KUKA KRL program: Inconel_dataset.src, Inconel_dataset.dat

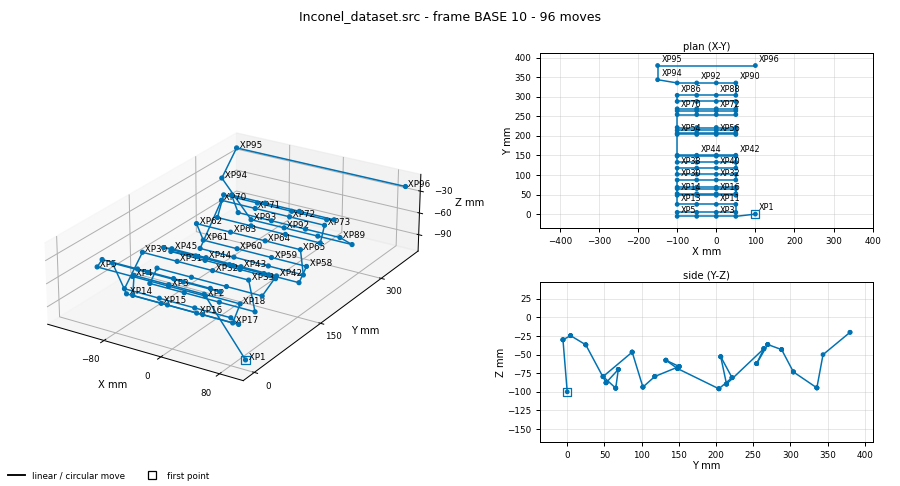
[picture p0: tool path of Inconel_dataset.src in frame BASE 10, 96 of 339 moves have a stored position in this frame; points joined in program order, loops and branches not executed]
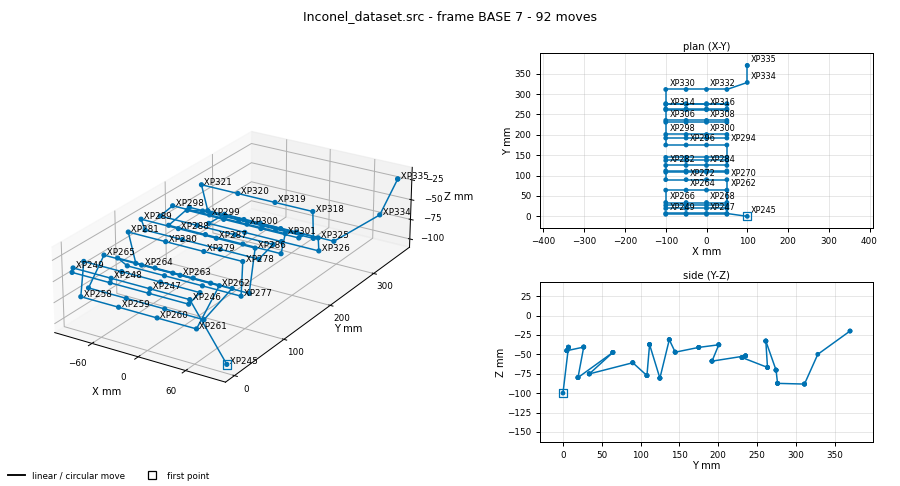
[picture p1: tool path of Inconel_dataset.src in frame BASE 7, 92 of 339 moves have a stored position in this frame; points joined in program order, loops and branches not executed]
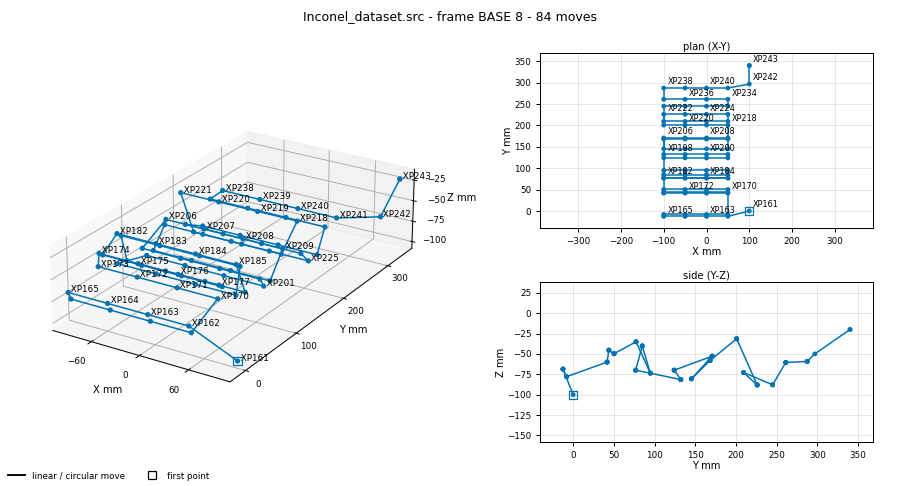
[picture p2: tool path of Inconel_dataset.src in frame BASE 8, 84 of 339 moves have a stored position in this frame; points joined in program order, loops and branches not executed]
--- Inconel_dataset.src ---
&ACCESS RVP1
&REL 1217
&PARAM WOPTRAJECTORYID = 2
&PARAM WOPTEMPLATENAME = WopCoreTemplatePath
&PARAM DISKPATH = KRC:\R1\Program\Working Paths
DEF  Inconel_dataset ( )

;FOLD INI
InitWopCoreSrc(#Init_Trajectory)
;ENDFOLD (INI)

;FOLD Manual mode
IF X_Rob_InManu THEN
;Write here the code executed only in manual mode

ENDIF
;ENDFOLD

X_Prod_En_Cours[2]=TRUE

;FOLD PTP PT_LoopPos1 Vel=10 % DEFAULT Tool[1]:Gun Base[0];%{PE}
;FOLD Parameters ;%{h}
;Params IlfProvider=kukaroboter.basistech.inlineforms.movement.old; Kuka.IsGlobalPoint=False; Kuka.PointName=PT_LoopPos1; Kuka.BlendingEnabled=False; Kuka.MoveDataPtpName=DEFAULT; Kuka.VelocityPtp=10; Kuka.CurrentCDSetIndex=0; Kuka.MovementParameterFieldEnabled=True; IlfCommand=PTP
;ENDFOLD
$BWDSTART = FALSE
PDAT_ACT = PDEFAULT
FDAT_ACT = FPT_LoopPos1
BAS(#PTP_PARAMS, 10.0)
SET_CD_PARAMS (0)
PTP XPT_LoopPos1
;ENDFOLD



;FOLD CHECK DAT-FILE GENERATION NUMBER
  IF APP_GENNUMBER <> 215375 THEN
    LOOP
      MsgQuit("InconsistenceSRCandDAT",,,,1)
      HALT
    ENDLOOP
  ENDIF
;ENDFOLD

;fold Jobinfo
;Job information: Inconel_dataset
;Product : 3.1.0.28784
;Date: 2026-09-10-16_16
;Project name: Inconel_dataset
;Author: Alhadi Zidan
;Company: CRITT-TJFU
;Division: CSAMProj
;Comment: Autogenerated CSAM Path
;endfold

; --- GLOBAL BLENDING OVERRIDES ---
$APO.CDIS = 1.0  ; Distance blending radius (mm)
$APO.CVEL = 100  ; Velocity blending (%)
$APO.CORI = 5.0  ; Orientation blending (degrees)
$ADVANCE = 5
;FOLD PTP P0 Vel=100 % P0 Tool[2] Base[10] ;%{PE}
;FOLD Parameters ;%{h}
;Params IlfProvider=kukaroboter.basistech.inlineforms.movement.old; Kuka.IsGlobalPoint=False; Kuka.PointName=P0; Kuka.BlendingEnabled=FALSE; Kuka.MoveDataName=PDATP0; Kuka.VelocityPath=100; Kuka.CurrentCDSetIndex=0; Kuka.MovementParameterFieldEnabled=True; IlfCommand=PTP
;ENDFOLD
$BWDSTART = FALSE
PDAT_ACT=PPDATP0
FDAT_ACT=FP0
BAS (#PTP_PARAMS,100)
SET_CD_PARAMS (0)
PTP XP0

;ENDFOLD
Routine_0()
Routine_1()
Routine_2()
Routine_3()
;FOLD PTP PT_LoopPos1 Vel=60 % DEFAULT Tool[1]:Gun Base[0];%{{PE}}
;FOLD Parameters ;%{{h}}
;Params IlfProvider=kukaroboter.basistech.inlineforms.movement.old; Kuka.IsGlobalPoint=False; Kuka.PointName=PT_LoopPos1; Kuka.BlendingEnabled=False; Kuka.MoveDataPtpName=DEFAULT; Kuka.VelocityPtp=10; Kuka.CurrentCDSetIndex=0; Kuka.MovementParameterFieldEnabled=True; IlfCommand=PTP
;ENDFOLD
$BWDSTART = FALSE
PDAT_ACT = PDEFAULT
FDAT_ACT = FPT_LoopPos1
BAS(#PTP_PARAMS, 60.0)
SET_CD_PARAMS (0)
PTP XPT_LoopPos1
;ENDFOLD
END

; --- Routine for substrate 0 ---
DEF Routine_0()
;FOLD LIN P1 CONT Vel=1.0 m/s CPDATP1 Tool[2] Base[10] ;%{PE}
;FOLD Parameters ;%{h}
;Params IlfProvider=kukaroboter.basistech.inlineforms.movement.old; Kuka.IsGlobalPoint=False; Kuka.PointName=P1; Kuka.BlendingEnabled=TRUE; Kuka.MoveDataName=CPDATP1; Kuka.VelocityPath=1.0; Kuka.CurrentCDSetIndex=0; Kuka.MovementParameterFieldEnabled=True; IlfCommand=LIN
;ENDFOLD
$BWDSTART = FALSE
LDAT_ACT=LCPDATP1
FDAT_ACT=FP1
BAS (#CP_PARAMS,1.0)
SET_CD_PARAMS (0)
LIN XP1 C_DIS

;ENDFOLD
;FOLD LIN P2 CONT Vel=0.116 m/s CPDATP2 Tool[2] Base[10] ;%{PE}
;FOLD Parameters ;%{h}
;Params IlfProvider=kukaroboter.basistech.inlineforms.movement.old; Kuka.IsGlobalPoint=False; Kuka.PointName=P2; Kuka.BlendingEnabled=TRUE; Kuka.MoveDataName=CPDATP2; Kuka.VelocityPath=0.116; Kuka.CurrentCDSetIndex=0; Kuka.MovementParameterFieldEnabled=True; IlfCommand=LIN
;ENDFOLD
$BWDSTART = FALSE
LDAT_ACT=LCPDATP2
FDAT_ACT=FP2
BAS (#CP_PARAMS,0.116)
SET_CD_PARAMS (0)
LIN XP2 C_DIS

;ENDFOLD
;FOLD LIN P3 CONT Vel=0.116 m/s CPDATP3 Tool[2] Base[10] ;%{PE}
;FOLD Parameters ;%{h}
;Params IlfProvider=kukaroboter.basistech.inlineforms.movement.old; Kuka.IsGlobalPoint=False; Kuka.PointName=P3; Kuka.BlendingEnabled=TRUE; Kuka.MoveDataName=CPDATP3; Kuka.VelocityPath=0.116; Kuka.CurrentCDSetIndex=0; Kuka.MovementParameterFieldEnabled=True; IlfCommand=LIN
;ENDFOLD
$BWDSTART = FALSE
LDAT_ACT=LCPDATP3
FDAT_ACT=FP3
BAS (#CP_PARAMS,0.116)
SET_CD_PARAMS (0)
LIN XP3 C_DIS

;ENDFOLD
;FOLD LIN P4 CONT Vel=0.116 m/s CPDATP4 Tool[2] Base[10] ;%{PE}
;FOLD Parameters ;%{h}
;Params IlfProvider=kukaroboter.basistech.inlineforms.movement.old; Kuka.IsGlobalPoint=False; Kuka.PointName=P4; Kuka.BlendingEnabled=TRUE; Kuka.MoveDataName=CPDATP4; Kuka.VelocityPath=0.116; Kuka.CurrentCDSetIndex=0; Kuka.MovementParameterFieldEnabled=True; IlfCommand=LIN
;ENDFOLD
$BWDSTART = FALSE
LDAT_ACT=LCPDATP4
FDAT_ACT=FP4
BAS (#CP_PARAMS,0.116)
SET_CD_PARAMS (0)
LIN XP4 C_DIS

;ENDFOLD
;FOLD LIN P5 CONT Vel=0.116 m/s CPDATP5 Tool[2] Base[10] ;%{PE}
;FOLD Parameters ;%{h}
;Params IlfProvider=kukaroboter.basistech.inlineforms.movement.old; Kuka.IsGlobalPoint=False; Kuka.PointName=P5; Kuka.BlendingEnabled=TRUE; Kuka.MoveDataName=CPDATP5; Kuka.VelocityPath=0.116; Kuka.CurrentCDSetIndex=0; Kuka.MovementParameterFieldEnabled=True; IlfCommand=LIN
;ENDFOLD
$BWDSTART = FALSE
LDAT_ACT=LCPDATP5
FDAT_ACT=FP5
BAS (#CP_PARAMS,0.116)
SET_CD_PARAMS (0)
LIN XP5 C_DIS

;ENDFOLD
;FOLD LIN P6 CONT Vel=0.099 m/s CPDATP6 Tool[2] Base[10] ;%{PE}
;FOLD Parameters ;%{h}
;Params IlfProvider=kukaroboter.basistech.inlineforms.movement.old; Kuka.IsGlobalPoint=False; Kuka.PointName=P6; Kuka.BlendingEnabled=TRUE; Kuka.MoveDataName=CPDATP6; Kuka.VelocityPath=0.099; Kuka.CurrentCDSetIndex=0; Kuka.MovementParameterFieldEnabled=True; IlfCommand=LIN
;ENDFOLD
$BWDSTART = FALSE
LDAT_ACT=LCPDATP6
FDAT_ACT=FP6
BAS (#CP_PARAMS,0.099)
SET_CD_PARAMS (0)
LIN XP6 C_DIS

;ENDFOLD
;FOLD LIN P7 CONT Vel=0.099 m/s CPDATP7 Tool[2] Base[10] ;%{PE}
;FOLD Parameters ;%{h}
;Params IlfProvider=kukaroboter.basistech.inlineforms.movement.old; Kuka.IsGlobalPoint=False; Kuka.PointName=P7; Kuka.BlendingEnabled=TRUE; Kuka.MoveDataName=CPDATP7; Kuka.VelocityPath=0.099; Kuka.CurrentCDSetIndex=0; Kuka.MovementParameterFieldEnabled=True; IlfCommand=LIN
;ENDFOLD
$BWDSTART = FALSE
LDAT_ACT=LCPDATP7
FDAT_ACT=FP7
BAS (#CP_PARAMS,0.099)
SET_CD_PARAMS (0)
LIN XP7 C_DIS

;ENDFOLD
;FOLD LIN P8 CONT Vel=0.099 m/s CPDATP8 Tool[2] Base[10] ;%{PE}
;FOLD Parameters ;%{h}
;Params IlfProvider=kukaroboter.basistech.inlineforms.movement.old; Kuka.IsGlobalPoint=False; Kuka.PointName=P8; Kuka.BlendingEnabled=TRUE; Kuka.MoveDataName=CPDATP8; Kuka.VelocityPath=0.099; Kuka.CurrentCDSetIndex=0; Kuka.MovementParameterFieldEnabled=True; IlfCommand=LIN
;ENDFOLD
$BWDSTART = FALSE
LDAT_ACT=LCPDATP8
FDAT_ACT=FP8
BAS (#CP_PARAMS,0.099)
SET_CD_PARAMS (0)
LIN XP8 C_DIS

;ENDFOLD
;FOLD LIN P9 CONT Vel=0.099 m/s CPDATP9 Tool[2] Base[10] ;%{PE}
;FOLD Parameters ;%{h}
;Params IlfProvider=kukaroboter.basistech.inlineforms.movement.old; Kuka.IsGlobalPoint=False; Kuka.PointName=P9; Kuka.BlendingEnabled=TRUE; Kuka.MoveDataName=CPDATP9; Kuka.VelocityPath=0.099; Kuka.CurrentCDSetIndex=0; Kuka.MovementParameterFieldEnabled=True; IlfCommand=LIN
;ENDFOLD
$BWDSTART = FALSE
LDAT_ACT=LCPDATP9
FDAT_ACT=FP9
BAS (#CP_PARAMS,0.099)
SET_CD_PARAMS (0)
LIN XP9 C_DIS

;ENDFOLD
;FOLD LIN P10 CONT Vel=0.075 m/s CPDATP10 Tool[2] Base[10] ;%{PE}
;FOLD Parameters ;%{h}
;Params IlfProvider=kukaroboter.basistech.inlineforms.movement.old; Kuka.IsGlobalPoint=False; Kuka.PointName=P10; Kuka.BlendingEnabled=TRUE; Kuka.MoveDataName=CPDATP10; Kuka.VelocityPath=0.075; Kuka.CurrentCDSetIndex=0; Kuka.MovementParameterFieldEnabled=True; IlfCommand=LIN
;ENDFOLD
$BWDSTART = FALSE
LDAT_ACT=LCPDATP10
FDAT_ACT=FP10
BAS (#CP_PARAMS,0.075)
SET_CD_PARAMS (0)
LIN XP10 C_DIS

;ENDFOLD
;FOLD LIN P11 CONT Vel=0.075 m/s CPDATP11 Tool[2] Base[10] ;%{PE}
;FOLD Parameters ;%{h}
;Params IlfProvider=kukaroboter.basistech.inlineforms.movement.old; Kuka.IsGlobalPoint=False; Kuka.PointName=P11; Kuka.BlendingEnabled=TRUE; Kuka.MoveDataName=CPDATP11; Kuka.VelocityPath=0.075; Kuka.CurrentCDSetIndex=0; Kuka.MovementParameterFieldEnabled=True; IlfCommand=LIN
;ENDFOLD
$BWDSTART = FALSE
LDAT_ACT=LCPDATP11
FDAT_ACT=FP11
BAS (#CP_PARAMS,0.075)
SET_CD_PARAMS (0)
LIN XP11 C_DIS

;ENDFOLD
;FOLD LIN P12 CONT Vel=0.075 m/s CPDATP12 Tool[2] Base[10] ;%{PE}
;FOLD Parameters ;%{h}
;Params IlfProvider=kukaroboter.basistech.inlineforms.movement.old; Kuka.IsGlobalPoint=False; Kuka.PointName=P12; Kuka.BlendingEnabled=TRUE; Kuka.MoveDataName=CPDATP12; Kuka.VelocityPath=0.075; Kuka.CurrentCDSetIndex=0; Kuka.MovementParameterFieldEnabled=True; IlfCommand=LIN
;ENDFOLD
$BWDSTART = FALSE
LDAT_ACT=LCPDATP12
FDAT_ACT=FP12
BAS (#CP_PARAMS,0.075)
SET_CD_PARAMS (0)
LIN XP12 C_DIS

;ENDFOLD
;FOLD LIN P13 CONT Vel=0.075 m/s CPDATP13 Tool[2] Base[10] ;%{PE}
;FOLD Parameters ;%{h}
;Params IlfProvider=kukaroboter.basistech.inlineforms.movement.old; Kuka.IsGlobalPoint=False; Kuka.PointName=P13; Kuka.BlendingEnabled=TRUE; Kuka.MoveDataName=CPDATP13; Kuka.VelocityPath=0.075; Kuka.CurrentCDSetIndex=0; Kuka.MovementParameterFieldEnabled=True; IlfCommand=LIN
;ENDFOLD
$BWDSTART = FALSE
LDAT_ACT=LCPDATP13
FDAT_ACT=FP13
BAS (#CP_PARAMS,0.075)
SET_CD_PARAMS (0)
LIN XP13 C_DIS

;ENDFOLD
;FOLD LIN P14 CONT Vel=0.113 m/s CPDATP14 Tool[2] Base[10] ;%{PE}
;FOLD Parameters ;%{h}
;Params IlfProvider=kukaroboter.basistech.inlineforms.movement.old; Kuka.IsGlobalPoint=False; Kuka.PointName=P14; Kuka.BlendingEnabled=TRUE; Kuka.MoveDataName=CPDATP14; Kuka.VelocityPath=0.113; Kuka.CurrentCDSetIndex=0; Kuka.MovementParameterFieldEnabled=True; IlfCommand=LIN
;ENDFOLD
$BWDSTART = FALSE
LDAT_ACT=LCPDATP14
FDAT_ACT=FP14
BAS (#CP_PARAMS,0.113)
SET_CD_PARAMS (0)
LIN XP14 C_DIS

;ENDFOLD
;FOLD LIN P15 CONT Vel=0.113 m/s CPDATP15 Tool[2] Base[10] ;%{PE}
;FOLD Parameters ;%{h}
;Params IlfProvider=kukaroboter.basistech.inlineforms.movement.old; Kuka.IsGlobalPoint=False; Kuka.PointName=P15; Kuka.BlendingEnabled=TRUE; Kuka.MoveDataName=CPDATP15; Kuka.VelocityPath=0.113; Kuka.CurrentCDSetIndex=0; Kuka.MovementParameterFieldEnabled=True; IlfCommand=LIN
;ENDFOLD
$BWDSTART = FALSE
LDAT_ACT=LCPDATP15
FDAT_ACT=FP15
BAS (#CP_PARAMS,0.113)
SET_CD_PARAMS (0)
LIN XP15 C_DIS

;ENDFOLD
;FOLD LIN P16 CONT Vel=0.113 m/s CPDATP16 Tool[2] Base[10] ;%{PE}
;FOLD Parameters ;%{h}
;Params IlfProvider=kukaroboter.basistech.inlineforms.movement.old; Kuka.IsGlobalPoint=False; Kuka.PointName=P16; Kuka.BlendingEnabled=TRUE; Kuka.MoveDataName=CPDATP16; Kuka.VelocityPath=0.113; Kuka.CurrentCDSetIndex=0; Kuka.MovementParameterFieldEnabled=True; IlfCommand=LIN
;ENDFOLD
$BWDSTART = FALSE
LDAT_ACT=LCPDATP16
FDAT_ACT=FP16
BAS (#CP_PARAMS,0.113)
SET_CD_PARAMS (0)
LIN XP16 C_DIS

;ENDFOLD
;FOLD LIN P17 CONT Vel=0.113 m/s CPDATP17 Tool[2] Base[10] ;%{PE}
;FOLD Parameters ;%{h}
;Params IlfProvider=kukaroboter.basistech.inlineforms.movement.old; Kuka.IsGlobalPoint=False; Kuka.PointName=P17; Kuka.BlendingEnabled=TRUE; Kuka.MoveDataName=CPDATP17; Kuka.VelocityPath=0.113; Kuka.CurrentCDSetIndex=0; Kuka.MovementParameterFieldEnabled=True; IlfCommand=LIN
;ENDFOLD
$BWDSTART = FALSE
LDAT_ACT=LCPDATP17
FDAT_ACT=FP17
BAS (#CP_PARAMS,0.113)
SET_CD_PARAMS (0)
LIN XP17 C_DIS

;ENDFOLD
;FOLD LIN P18 CONT Vel=0.086 m/s CPDATP18 Tool[2] Base[10] ;%{PE}
;FOLD Parameters ;%{h}
;Params IlfProvider=kukaroboter.basistech.inlineforms.movement.old; Kuka.IsGlobalPoint=False; Kuka.PointName=P18; Kuka.BlendingEnabled=TRUE; Kuka.MoveDataName=CPDATP18; Kuka.VelocityPath=0.086; Kuka.CurrentCDSetIndex=0; Kuka.MovementParameterFieldEnabled=True; IlfCommand=LIN
;ENDFOLD
$BWDSTART = FALSE
LDAT_ACT=LCPDATP18
FDAT_ACT=FP18
BAS (#CP_PARAMS,0.086)
SET_CD_PARAMS (0)
LIN XP18 C_DIS

;ENDFOLD
;FOLD LIN P19 CONT Vel=0.086 m/s CPDATP19 Tool[2] Base[10] ;%{PE}
;FOLD Parameters ;%{h}
;Params IlfProvider=kukaroboter.basistech.inlineforms.movement.old; Kuka.IsGlobalPoint=False; Kuka.PointName=P19; Kuka.BlendingEnabled=TRUE; Kuka.MoveDataName=CPDATP19; Kuka.VelocityPath=0.086; Kuka.CurrentCDSetIndex=0; Kuka.MovementParameterFieldEnabled=True; IlfCommand=LIN
;ENDFOLD
$BWDSTART = FALSE
LDAT_ACT=LCPDATP19
FDAT_ACT=FP19
BAS (#CP_PARAMS,0.086)
SET_CD_PARAMS (0)
LIN XP19 C_DIS

;ENDFOLD
;FOLD LIN P20 CONT Vel=0.086 m/s CPDATP20 Tool[2] Base[10] ;%{PE}
;FOLD Parameters ;%{h}
;Params IlfProvider=kukaroboter.basistech.inlineforms.movement.old; Kuka.IsGlobalPoint=False; Kuka.PointName=P20; Kuka.BlendingEnabled=TRUE; Kuka.MoveDataName=CPDATP20; Kuka.VelocityPath=0.086; Kuka.CurrentCDSetIndex=0; Kuka.MovementParameterFieldEnabled=True; IlfCommand=LIN
;ENDFOLD
$BWDSTART = FALSE
LDAT_ACT=LCPDATP20
FDAT_ACT=FP20
BAS (#CP_PARAMS,0.086)
SET_CD_PARAMS (0)
LIN XP20 C_DIS

;ENDFOLD
;FOLD LIN P21 CONT Vel=0.086 m/s CPDATP21 Tool[2] Base[10] ;%{PE}
;FOLD Parameters ;%{h}
;Params IlfProvider=kukaroboter.basistech.inlineforms.movement.old; Kuka.IsGlobalPoint=False; Kuka.PointName=P21; Kuka.BlendingEnabled=TRUE; Kuka.MoveDataName=CPDATP21; Kuka.VelocityPath=0.086; Kuka.CurrentCDSetIndex=0; Kuka.MovementParameterFieldEnabled=True; IlfCommand=LIN
;ENDFOLD
$BWDSTART = FALSE
LDAT_ACT=LCPDATP21
FDAT_ACT=FP21
BAS (#CP_PARAMS,0.086)
SET_CD_PARAMS (0)
LIN XP21 C_DIS

;ENDFOLD
;FOLD LIN P22 CONT Vel=0.073 m/s CPDATP22 Tool[2] Base[10] ;%{PE}
;FOLD Parameters ;%{h}
;Params IlfProvider=kukaroboter.basistech.inlineforms.movement.old; Kuka.IsGlobalPoint=False; Kuka.PointName=P22; Kuka.BlendingEnabled=TRUE; Kuka.MoveDataName=CPDATP22; Kuka.VelocityPath=0.073; Kuka.CurrentCDSetIndex=0; Kuka.MovementParameterFieldEnabled=True; IlfCommand=LIN
;ENDFOLD
$BWDSTART = FALSE
LDAT_ACT=LCPDATP22
FDAT_ACT=FP22
BAS (#CP_PARAMS,0.073)
SET_CD_PARAMS (0)
LIN XP22 C_DIS

;ENDFOLD
;FOLD LIN P23 CONT Vel=0.073 m/s CPDATP23 Tool[2] Base[10] ;%{PE}
;FOLD Parameters ;%{h}
;Params IlfProvider=kukaroboter.basistech.inlineforms.movement.old; Kuka.IsGlobalPoint=False; Kuka.PointName=P23; Kuka.BlendingEnabled=TRUE; Kuka.MoveDataName=CPDATP23; Kuka.VelocityPath=0.073; Kuka.CurrentCDSetIndex=0; Kuka.MovementParameterFieldEnabled=True; IlfCommand=LIN
;ENDFOLD
$BWDSTART = FALSE
LDAT_ACT=LCPDATP23
FDAT_ACT=FP23
BAS (#CP_PARAMS,0.073)
SET_CD_PARAMS (0)
LIN XP23 C_DIS

;ENDFOLD
;FOLD LIN P24 CONT Vel=0.073 m/s CPDATP24 Tool[2] Base[10] ;%{PE}
;FOLD Parameters ;%{h}
;Params IlfProvider=kukaroboter.basistech.inlineforms.movement.old; Kuka.IsGlobalPoint=False; Kuka.PointName=P24; Kuka.BlendingEnabled=TRUE; Kuka.MoveDataName=CPDATP24; Kuka.VelocityPath=0.073; Kuka.CurrentCDSetIndex=0; Kuka.MovementParameterFieldEnabled=True; IlfCommand=LIN
;ENDFOLD
$BWDSTART = FALSE
LDAT_ACT=LCPDATP24
FDAT_ACT=FP24
BAS (#CP_PARAMS,0.073)
SET_CD_PARAMS (0)
LIN XP24 C_DIS

;ENDFOLD
;FOLD LIN P25 CONT Vel=0.073 m/s CPDATP25 Tool[2] Base[10] ;%{PE}
;FOLD Parameters ;%{h}
;Params IlfProvider=kukaroboter.basistech.inlineforms.movement.old; Kuka.IsGlobalPoint=False; Kuka.PointName=P25; Kuka.BlendingEnabled=TRUE; Kuka.MoveDataName=CPDATP25; Kuka.VelocityPath=0.073; Kuka.CurrentCDSetIndex=0; Kuka.MovementParameterFieldEnabled=True; IlfCommand=LIN
;ENDFOLD
$BWDSTART = FALSE
LDAT_ACT=LCPDATP25
FDAT_ACT=FP25
BAS (#CP_PARAMS,0.073)
SET_CD_PARAMS (0)
LIN XP25 C_DIS

;ENDFOLD
;FOLD LIN P26 CONT Vel=0.137 m/s CPDATP26 Tool[2] Base[10] ;%{PE}
;FOLD Parameters ;%{h}
;Params IlfProvider=kukaroboter.basistech.inlineforms.movement.old; Kuka.IsGlobalPoint=False; Kuka.PointName=P26; Kuka.BlendingEnabled=TRUE; Kuka.MoveDataName=CPDATP26; Kuka.VelocityPath=0.137; Kuka.CurrentCDSetIndex=0; Kuka.MovementParameterFieldEnabled=True; IlfCommand=LIN
;ENDFOLD
$BWDSTART = FALSE
LDAT_ACT=LCPDATP26
FDAT_ACT=FP26
BAS (#CP_PARAMS,0.137)
SET_CD_PARAMS (0)
LIN XP26 C_DIS

;ENDFOLD
;FOLD LIN P27 CONT Vel=0.137 m/s CPDATP27 Tool[2] Base[10] ;%{PE}
;FOLD Parameters ;%{h}
;Params IlfProvider=kukaroboter.basistech.inlineforms.movement.old; Kuka.IsGlobalPoint=False; Kuka.PointName=P27; Kuka.BlendingEnabled=TRUE; Kuka.MoveDataName=CPDATP27; Kuka.VelocityPath=0.137; Kuka.CurrentCDSetIndex=0; Kuka.MovementParameterFieldEnabled=True; IlfCommand=LIN
;ENDFOLD
$BWDSTART = FALSE
LDAT_ACT=LCPDATP27
FDAT_ACT=FP27
BAS (#CP_PARAMS,0.137)
SET_CD_PARAMS (0)
LIN XP27 C_DIS

;ENDFOLD
;FOLD LIN P28 CONT Vel=0.137 m/s CPDATP28 Tool[2] Base[10] ;%{PE}
;FOLD Parameters ;%{h}
;Params IlfProvider=kukaroboter.basistech.inlineforms.movement.old; Kuka.IsGlobalPoint=False; Kuka.PointName=P28; Kuka.BlendingEnabled=TRUE; Kuka.MoveDataName=CPDATP28; Kuka.VelocityPath=0.137; Kuka.CurrentCDSetIndex=0; Kuka.MovementParameterFieldEnabled=True; IlfCommand=LIN
;ENDFOLD
$BWDSTART = FALSE
LDAT_ACT=LCPDATP28
FDAT_ACT=FP28
BAS (#CP_PARAMS,0.137)
SET_CD_PARAMS (0)
LIN XP28 C_DIS

;ENDFOLD
;FOLD LIN P29 CONT Vel=0.137 m/s CPDATP29 Tool[2] Base[10] ;%{PE}
;FOLD Parameters ;%{h}
;Params IlfProvider=kukaroboter.basistech.inlineforms.movement.old; Kuka.IsGlobalPoint=False; Kuka.PointName=P29; Kuka.BlendingEnabled=TRUE; Kuka.MoveDataName=CPDATP29; Kuka.VelocityPath=0.137; Kuka.CurrentCDSetIndex=0; Kuka.MovementParameterFieldEnabled=True; IlfCommand=LIN
;ENDFOLD
$BWDSTART = FALSE
LDAT_ACT=LCPDATP29
FDAT_ACT=FP29
BAS (#CP_PARAMS,0.137)
SET_CD_PARAMS (0)
LIN XP29 C_DIS

;ENDFOLD
;FOLD LIN P30 CONT Vel=0.082 m/s CPDATP30 Tool[2] Base[10] ;%{PE}
;FOLD Parameters ;%{h}
;Params IlfProvider=kukaroboter.basistech.inlineforms.movement.old; Kuka.IsGlobalPoint=False; Kuka.PointName=P30; Kuka.BlendingEnabled=TRUE; Kuka.MoveDataName=CPDATP30; Kuka.VelocityPath=0.082; Kuka.CurrentCDSetIndex=0; Kuka.MovementParameterFieldEnabled=True; IlfCommand=LIN
;ENDFOLD
$BWDSTART = FALSE
LDAT_ACT=LCPDATP30
FDAT_ACT=FP30
BAS (#CP_PARAMS,0.082)
SET_CD_PARAMS (0)
LIN XP30 C_DIS

;ENDFOLD
;FOLD LIN P31 CONT Vel=0.082 m/s CPDATP31 Tool[2] Base[10] ;%{PE}
;FOLD Parameters ;%{h}
;Params IlfProvider=kukaroboter.basistech.inlineforms.movement.old; Kuka.IsGlobalPoint=False; Kuka.PointName=P31; Kuka.BlendingEnabled=TRUE; Kuka.MoveDataName=CPDATP31; Kuka.VelocityPath=0.082; Kuka.CurrentCDSetIndex=0; Kuka.MovementParameterFieldEnabled=True; IlfCommand=LIN
;ENDFOLD
$BWDSTART = FALSE
LDAT_ACT=LCPDATP31
FDAT_ACT=FP31
BAS (#CP_PARAMS,0.082)
SET_CD_PARAMS (0)
LIN XP31 C_DIS

;ENDFOLD
;FOLD LIN P32 CONT Vel=0.082 m/s CPDATP32 Tool[2] Base[10] ;%{PE}
;FOLD Parameters ;%{h}
;Params IlfProvider=kukaroboter.basistech.inlineforms.movement.old; Kuka.IsGlobalPoint=False; Kuka.PointName=P32; Kuka.BlendingEnabled=TRUE; Kuka.MoveDataName=CPDATP32; Kuka.VelocityPath=0.082; Kuka.CurrentCDSetIndex=0; Kuka.MovementParameterFieldEnabled=True; IlfCommand=LIN
;ENDFOLD
$BWDSTART = FALSE
LDAT_ACT=LCPDATP32
FDAT_ACT=FP32
BAS (#CP_PARAMS,0.082)
SET_CD_PARAMS (0)
LIN XP32 C_DIS

;ENDFOLD
;FOLD LIN P33 CONT Vel=0.082 m/s CPDATP33 Tool[2] Base[10] ;%{PE}
;FOLD Parameters ;%{h}
;Params IlfProvider=kukaroboter.basistech.inlineforms.movement.old; Kuka.IsGlobalPoint=False; Kuka.PointName=P33; Kuka.BlendingEnabled=TRUE; Kuka.MoveDataName=CPDATP33; Kuka.VelocityPath=0.082; Kuka.CurrentCDSetIndex=0; Kuka.MovementParameterFieldEnabled=True; IlfCommand=LIN
;ENDFOLD
$BWDSTART = FALSE
LDAT_ACT=LCPDATP33
FDAT_ACT=FP33
BAS (#CP_PARAMS,0.082)
SET_CD_PARAMS (0)
LIN XP33 C_DIS

;ENDFOLD
;FOLD LIN P34 CONT Vel=0.086 m/s CPDATP34 Tool[2] Base[10] ;%{PE}
;FOLD Parameters ;%{h}
;Params IlfProvider=kukaroboter.basistech.inlineforms.movement.old; Kuka.IsGlobalPoint=False; Kuka.PointName=P34; Kuka.BlendingEnabled=TRUE; Kuka.MoveDataName=CPDATP34; Kuka.VelocityPath=0.086; Kuka.CurrentCDSetIndex=0; Kuka.MovementParameterFieldEnabled=True; IlfCommand=LIN
;ENDFOLD
$BWDSTART = FALSE
LDAT_ACT=LCPDATP34
FDAT_ACT=FP34
BAS (#CP_PARAMS,0.086)
SET_CD_PARAMS (0)
LIN XP34 C_DIS

;ENDFOLD
;FOLD LIN P35 CONT Vel=0.086 m/s CPDATP35 Tool[2] Base[10] ;%{PE}
;FOLD Parameters ;%{h}
;Params IlfProvider=kukaroboter.basistech.inlineforms.movement.old; Kuka.IsGlobalPoint=False; Kuka.PointName=P35; Kuka.BlendingEnabled=TRUE; Kuka.MoveDataName=CPDATP35; Kuka.VelocityPath=0.086; Kuka.CurrentCDSetIndex=0; Kuka.MovementParameterFieldEnabled=True; IlfCommand=LIN
;ENDFOLD
$BWDSTART = FALSE
LDAT_ACT=LCPDATP35
FDAT_ACT=FP35
BAS (#CP_PARAMS,0.086)
SET_CD_PARAMS (0)
LIN XP35 C_DIS

;ENDFOLD
;FOLD LIN P36 CONT Vel=0.086 m/s CPDATP36 Tool[2] Base[10] ;%{PE}
;FOLD Parameters ;%{h}
;Params IlfProvider=kukaroboter.basistech.inlineforms.movement.old; Kuka.IsGlobalPoint=False; Kuka.PointName=P36; Kuka.BlendingEnabled=TRUE; Kuka.MoveDataName=CPDATP36; Kuka.VelocityPath=0.086; Kuka.CurrentCDSetIndex=0; Kuka.MovementParameterFieldEnabled=True; IlfCommand=LIN
;ENDFOLD
$BWDSTART = FALSE
LDAT_ACT=LCPDATP36
FDAT_ACT=FP36
BAS (#CP_PARAMS,0.086)
SET_CD_PARAMS (0)
LIN XP36 C_DIS

;ENDFOLD
;FOLD LIN P37 CONT Vel=0.086 m/s CPDATP37 Tool[2] Base[10] ;%{PE}
;FOLD Parameters ;%{h}
;Params IlfProvider=kukaroboter.basistech.inlineforms.movement.old; Kuka.IsGlobalPoint=False; Kuka.PointName=P37; Kuka.BlendingEnabled=TRUE; Kuka.MoveDataName=CPDATP37; Kuka.VelocityPath=0.086; Kuka.CurrentCDSetIndex=0; Kuka.MovementParameterFieldEnabled=True; IlfCommand=LIN
;ENDFOLD
$BWDSTART = FALSE
LDAT_ACT=LCPDATP37
FDAT_ACT=FP37
BAS (#CP_PARAMS,0.086)
SET_CD_PARAMS (0)
LIN XP37 C_DIS

;ENDFOLD
;FOLD LIN P38 CONT Vel=0.097 m/s CPDATP38 Tool[2] Base[10] ;%{PE}
;FOLD Parameters ;%{h}
;Params IlfProvider=kukaroboter.basistech.inlineforms.movement.old; Kuka.IsGlobalPoint=False; Kuka.PointName=P38; Kuka.BlendingEnabled=TRUE; Kuka.MoveDataName=CPDATP38; Kuka.VelocityPath=0.097; Kuka.CurrentCDSetIndex=0; Kuka.MovementParameterFieldEnabled=True; IlfCommand=LIN
;ENDFOLD
$BWDSTART = FALSE
LDAT_ACT=LCPDATP38
FDAT_ACT=FP38
BAS (#CP_PARAMS,0.097)
SET_CD_PARAMS (0)
LIN XP38 C_DIS

;ENDFOLD
;FOLD LIN P39 CONT Vel=0.097 m/s CPDATP39 Tool[2] Base[10] ;%{PE}
;FOLD Parameters ;%{h}
;Params IlfProvider=kukaroboter.basistech.inlineforms.movement.old; Kuka.IsGlobalPoint=False; Kuka.PointName=P39; Kuka.BlendingEnabled=TRUE; Kuka.MoveDataName=CPDATP39; Kuka.VelocityPath=0.097; Kuka.CurrentCDSetIndex=0; Kuka.MovementParameterFieldEnabled=True; IlfCommand=LIN
;ENDFOLD
$BWDSTART = FALSE
LDAT_ACT=LCPDATP39
FDAT_ACT=FP39
BAS (#CP_PARAMS,0.097)
SET_CD_PARAMS (0)
LIN XP39 C_DIS

;ENDFOLD
;FOLD LIN P40 CONT Vel=0.097 m/s CPDATP40 Tool[2] Base[10] ;%{PE}
;FOLD Parameters ;%{h}
;Params IlfProvider=kukaroboter.basistech.inlineforms.movement.old; Kuka.IsGlobalPoint=False; Kuka.PointName=P40; Kuka.BlendingEnabled=TRUE; Kuka.MoveDataName=CPDATP40; Kuka.VelocityPath=0.097; Kuka.CurrentCDSetIndex=0; Kuka.MovementParameterFieldEnabled=True; IlfCommand=LIN
;ENDFOLD
$BWDSTART = FALSE
LDAT_ACT=LCPDATP40
FDAT_ACT=FP40
BAS (#CP_PARAMS,0.097)
SET_CD_PARAMS (0)
LIN XP40 C_DIS

;ENDFOLD
;FOLD LIN P41 CONT Vel=0.097 m/s CPDATP41 Tool[2] Base[10] ;%{PE}
;FOLD Parameters ;%{h}
;Params IlfProvider=kukaroboter.basistech.inlineforms.movement.old; Kuka.IsGlobalPoint=False; Kuka.PointName=P41; Kuka.BlendingEnabled=TRUE; Kuka.MoveDataName=CPDATP41; Kuka.VelocityPath=0.097; Kuka.CurrentCDSetIndex=0; Kuka.MovementParameterFieldEnabled=True; IlfCommand=LIN
;ENDFOLD
$BWDSTART = FALSE
LDAT_ACT=LCPDATP41
FDAT_ACT=FP41
BAS (#CP_PARAMS,0.097)
SET_CD_PARAMS (0)
LIN XP41 C_DIS

;ENDFOLD
;FOLD LIN P42 CONT Vel=0.136 m/s CPDATP42 Tool[2] Base[10] ;%{PE}
;FOLD Parameters ;%{h}
;Params IlfProvider=kukaroboter.basistech.inlineforms.movement.old; Kuka.IsGlobalPoint=False; Kuka.PointName=P42; Kuka.BlendingEnabled=TRUE; Kuka.MoveDataName=CPDATP42; Kuka.VelocityPath=0.136; Kuka.CurrentCDSetIndex=0; Kuka.MovementParameterFieldEnabled=True; IlfCommand=LIN
;ENDFOLD
$BWDSTART = FALSE
LDAT_ACT=LCPDATP42
FDAT_ACT=FP42
BAS (#CP_PARAMS,0.136)
SET_CD_PARAMS (0)
LIN XP42 C_DIS

;ENDFOLD
;FOLD LIN P43 CONT Vel=0.136 m/s CPDATP43 Tool[2] Base[10] ;%{PE}
;FOLD Parameters ;%{h}
;Params IlfProvider=kukaroboter.basistech.inlineforms.movement.old; Kuka.IsGlobalPoint=False; Kuka.PointName=P43; Kuka.BlendingEnabled=TRUE; Kuka.MoveDataName=CPDATP43; Kuka.VelocityPath=0.136; Kuka.CurrentCDSetIndex=0; Kuka.MovementParameterFieldEnabled=True; IlfCommand=LIN
;ENDFOLD
$BWDSTART = FALSE
LDAT_ACT=LCPDATP43
FDAT_ACT=FP43
BAS (#CP_PARAMS,0.136)
SET_CD_PARAMS (0)
LIN XP43 C_DIS

;ENDFOLD
;FOLD LIN P44 CONT Vel=0.136 m/s CPDATP44 Tool[2] Base[10] ;%{PE}
;FOLD Parameters ;%{h}
;Params IlfProvider=kukaroboter.basistech.inlineforms.movement.old; Kuka.IsGlobalPoint=False; Kuka.PointName=P44; Kuka.BlendingEnabled=TRUE; Kuka.MoveDataName=CPDATP44; Kuka.VelocityPath=0.136; Kuka.CurrentCDSetIndex=0; Kuka.MovementParameterFieldEnabled=True; IlfCommand=LIN
;ENDFOLD
$BWDSTART = FALSE
LDAT_ACT=LCPDATP44
FDAT_ACT=FP44
BAS (#CP_PARAMS,0.136)
SET_CD_PARAMS (0)
LIN XP44 C_DIS

;ENDFOLD
;FOLD LIN P45 CONT Vel=0.136 m/s CPDATP45 Tool[2] Base[10] ;%{PE}
;FOLD Parameters ;%{h}
;Params IlfProvider=kukaroboter.basistech.inlineforms.movement.old; Kuka.IsGlobalPoint=False; Kuka.PointName=P45; Kuka.BlendingEnabled=TRUE; Kuka.MoveDataName=CPDATP45; Kuka.VelocityPath=0.136; Kuka.CurrentCDSetIndex=0; Kuka.MovementParameterFieldEnabled=True; IlfCommand=LIN
;ENDFOLD
$BWDSTART = FALSE
LDAT_ACT=LCPDATP45
FDAT_ACT=FP45
BAS (#CP_PARAMS,0.136)
SET_CD_PARAMS (0)
LIN XP45 C_DIS

;ENDFOLD
;FOLD LIN P46 CONT Vel=0.107 m/s CPDATP46 Tool[2] Base[10] ;%{PE}
;FOLD Parameters ;%{h}
;Params IlfProvider=kukaroboter.basistech.inlineforms.movement.old; Kuka.IsGlobalPoint=False; Kuka.PointName=P46; Kuka.BlendingEnabled=TRUE; Kuka.MoveDataName=CPDATP46; Kuka.VelocityPath=0.107; Kuka.CurrentCDSetIndex=0; Kuka.MovementParameterFieldEnabled=True; IlfCommand=LIN
;ENDFOLD
$BWDSTART = FALSE
LDAT_ACT=LCPDATP46
FDAT_ACT=FP46
BAS (#CP_PARAMS,0.107)
SET_CD_PARAMS (0)
LIN XP46 C_DIS

;ENDFOLD
;FOLD LIN P47 CONT Vel=0.107 m/s CPDATP47 Tool[2] Base[10] ;%{PE}
;FOLD Parameters ;%{h}
;Params IlfProvider=kukaroboter.basistech.inlineforms.movement.old; Kuka.IsGlobalPoint=False; Kuka.PointName=P47; Kuka.BlendingEnabled=TRUE; Kuka.MoveDataName=CPDATP47; Kuka.VelocityPath=0.107; Kuka.CurrentCDSetIndex=0; Kuka.MovementParameterFieldEnabled=True; IlfCommand=LIN
;ENDFOLD
$BWDSTART = FALSE
LDAT_ACT=LCPDATP47
FDAT_ACT=FP47
BAS (#CP_PARAMS,0.107)
SET_CD_PARAMS (0)
LIN XP47 C_DIS

;ENDFOLD
;FOLD LIN P48 CONT Vel=0.107 m/s CPDATP48 Tool[2] Base[10] ;%{PE}
;FOLD Parameters ;%{h}
;Params IlfProvider=kukaroboter.basistech.inlineforms.movement.old; Kuka.IsGlobalPoint=False; Kuka.PointName=P48; Kuka.BlendingEnabled=TRUE; Kuka.MoveDataName=CPDATP48; Kuka.VelocityPath=0.107; Kuka.CurrentCDSetIndex=0; Kuka.MovementParameterFieldEnabled=True; IlfCommand=LIN
;ENDFOLD
$BWDSTART = FALSE
LDAT_ACT=LCPDATP48
FDAT_ACT=FP48
BAS (#CP_PARAMS,0.107)
SET_CD_PARAMS (0)
LIN XP48 C_DIS

;ENDFOLD
;FOLD LIN P49 CONT Vel=0.107 m/s CPDATP49 Tool[2] Base[10] ;%{PE}
;FOLD Parameters ;%{h}
;Params IlfProvider=kukaroboter.basistech.inlineforms.movement.old; Kuka.IsGlobalPoint=False; Kuka.PointName=P49; Kuka.BlendingEnabled=TRUE; Kuka.MoveDataName=CPDATP49; Kuka.VelocityPath=0.107; Kuka.CurrentCDSetIndex=0; Kuka.MovementParameterFieldEnabled=True; IlfCommand=LIN
;ENDFOLD
$BWDSTART = FALSE
LDAT_ACT=LCPDATP49
FDAT_ACT=FP49
BAS (#CP_PARAMS,0.107)
SET_CD_PARAMS (0)
LIN XP49 C_DIS

;ENDFOLD
;FOLD LIN P50 CONT Vel=0.09 m/s CPDATP50 Tool[2] Base[10] ;%{PE}
;FOLD Parameters ;%{h}
;Params IlfProvider=kukaroboter.basistech.inlineforms.movement.old; Kuka.IsGlobalPoint=False; Kuka.PointName=P50; Kuka.BlendingEnabled=TRUE; Kuka.MoveDataName=CPDATP50; Kuka.VelocityPath=0.09; Kuka.CurrentCDSetIndex=0; Kuka.MovementParameterFieldEnabled=True; IlfCommand=LIN
;ENDFOLD
$BWDSTART = FALSE
LDAT_ACT=LCPDATP50
FDAT_ACT=FP50
BAS (#CP_PARAMS,0.09)
SET_CD_PARAMS (0)
LIN XP50 C_DIS

;ENDFOLD
;FOLD LIN P51 CONT Vel=0.09 m/s CPDATP51 Tool[2] Base[10] ;%{PE}
;FOLD Parameters ;%{h}
;Params IlfProvider=kukaroboter.basistech.inlineforms.movement.old; Kuka.IsGlobalPoint=False; Kuka.PointName=P51; Kuka.BlendingEnabled=TRUE; Kuka.MoveDataName=CPDATP51; Kuka.VelocityPath=0.09; Kuka.CurrentCDSetIndex=0; Kuka.MovementParameterFieldEnabled=True; IlfCommand=LIN
;ENDFOLD
$BWDSTART = FALSE
LDAT_ACT=LCPDATP51
FDAT_ACT=FP51
BAS (#CP_PARAMS,0.09)
SET_CD_PARAMS (0)
LIN XP51 C_DIS

;ENDFOLD
;FOLD LIN P52 CONT Vel=0.09 m/s CPDATP52 Tool[2] Base[10] ;%{PE}
;FOLD Parameters ;%{h}
;Params IlfProvider=kukaroboter.basistech.inlineforms.movement.old; Kuka.IsGlobalPoint=False; Kuka.PointName=P52; Kuka.BlendingEnabled=TRUE; Kuka.MoveDataName=CPDATP52; Kuka.VelocityPath=0.09; Kuka.CurrentCDSetIndex=0; Kuka.MovementParameterFieldEnabled=True; IlfCommand=LIN
;ENDFOLD
$BWDSTART = FALSE
LDAT_ACT=LCPDATP52
FDAT_ACT=FP52
BAS (#CP_PARAMS,0.09)
SET_CD_PARAMS (0)
LIN XP52 C_DIS

;ENDFOLD
;FOLD LIN P53 CONT Vel=0.09 m/s CPDATP53 Tool[2] Base[10] ;%{PE}
;FOLD Parameters ;%{h}
;Params IlfProvider=kukaroboter.basistech.inlineforms.movement.old; Kuka.IsGlobalPoint=False; Kuka.PointName=P53; Kuka.BlendingEnabled=TRUE; Kuka.MoveDataName=CPDATP53; Kuka.VelocityPath=0.09; Kuka.CurrentCDSetIndex=0; Kuka.MovementParameterFieldEnabled=True; IlfCommand=LIN
;ENDFOLD
$BWDSTART = FALSE
LDAT_ACT=LCPDATP53
FDAT_ACT=FP53
BAS (#CP_PARAMS,0.09)
SET_CD_PARAMS (0)
LIN XP53 C_DIS

;ENDFOLD
;FOLD LIN P54 CONT Vel=0.132 m/s CPDATP54 Tool[2] Base[10] ;%{PE}
;FOLD Parameters ;%{h}
;Params IlfProvider=kukaroboter.basistech.inlineforms.movement.old; Kuka.IsGlobalPoint=False; Kuka.PointName=P54; Kuka.BlendingEnabled=TRUE; Kuka.MoveDataName=CPDATP54; Kuka.VelocityPath=0.132; Kuka.CurrentCDSetIndex=0; Kuka.MovementParameterFieldEnabled=True; IlfCommand=LIN
;ENDFOLD
$BWDSTART = FALSE
LDAT_ACT=LCPDATP54
FDAT_ACT=FP54
BAS (#CP_PARAMS,0.132)
SET_CD_PARAMS (0)
LIN XP54 C_DIS

;ENDFOLD
;FOLD LIN P55 CONT Vel=0.132 m/s CPDATP55 Tool[2] Base[10] ;%{PE}
;FOLD Parameters ;%{h}
;Params IlfProvider=kukaroboter.basistech.inlineforms.movement.old; Kuka.IsGlobalPoint=False; Kuka.PointName=P55; Kuka.BlendingEnabled=TRUE; Kuka.MoveDataName=CPDATP55; Kuka.VelocityPath=0.132; Kuka.CurrentCDSetIndex=0; Kuka.MovementParameterFieldEnabled=True; IlfCommand=LIN
;ENDFOLD
$BWDSTART = FALSE
LDAT_ACT=LCPDATP55
FDAT_ACT=FP55
BAS (#CP_PARAMS,0.132)
SET_CD_PARAMS (0)
LIN XP55 C_DIS

;ENDFOLD
;FOLD LIN P56 CONT Vel=0.132 m/s CPDATP56 Tool[2] Base[10] ;%{PE}
;FOLD Parameters ;%{h}
;Params IlfProvider=kukaroboter.basistech.inlineforms.movement.old; Kuka.IsGlobalPoint=False; Kuka.PointName=P56; Kuka.BlendingEnabled=TRUE; Kuka.MoveDataName=CPDATP56; Kuka.VelocityPath=0.132; Kuka.CurrentCDSetIndex=0; Kuka.MovementParameterFieldEnabled=True; IlfCommand=LIN
;ENDFOLD
$BWDSTART = FALSE
LDAT_ACT=LCPDATP56
FDAT_ACT=FP56
BAS (#CP_PARAMS,0.132)
SET_CD_PARAMS (0)
LIN XP56 C_DIS

;ENDFOLD
;FOLD LIN P57 CONT Vel=0.132 m/s CPDATP57 Tool[2] Base[10] ;%{PE}
;FOLD Parameters ;%{h}
;Params IlfProvider=kukaroboter.basistech.inlineforms.movement.old; Kuka.IsGlobalPoint=False; Kuka.PointName=P57; Kuka.BlendingEnabled=TRUE; Kuka.MoveDataName=CPDATP57; Kuka.VelocityPath=0.132; Kuka.CurrentCDSetIndex=0; Kuka.MovementParameterFieldEnabled=True; IlfCommand=LIN
;ENDFOLD
$BWDSTART = FALSE
LDAT_ACT=LCPDATP57
FDAT_ACT=FP57
BAS (#CP_PARAMS,0.132)
SET_CD_PARAMS (0)
LIN XP57 C_DIS

;ENDFOLD
;FOLD LIN P58 CONT Vel=0.068 m/s CPDATP58 Tool[2] Base[10] ;%{PE}
;FOLD Parameters ;%{h}
;Params IlfProvider=kukaroboter.basistech.inlineforms.movement.old; Kuka.IsGlobalPoint=False; Kuka.PointName=P58; Kuka.BlendingEnabled=TRUE; Kuka.MoveDataName=CPDATP58; Kuka.VelocityPath=0.068; Kuka.CurrentCDSetIndex=0; Kuka.MovementParameterFieldEnabled=True; IlfCommand=LIN
;ENDFOLD
$BWDSTART = FALSE
LDAT_ACT=LCPDATP58
FDAT_ACT=FP58
BAS (#CP_PARAMS,0.068)
SET_CD_PARAMS (0)
LIN XP58 C_DIS

;ENDFOLD
;FOLD LIN P59 CONT Vel=0.068 m/s CPDATP59 Tool[2] Base[10] ;%{PE}
;FOLD Parameters ;%{h}
;Params IlfProvider=kukaroboter.basistech.inlineforms.movement.old; Kuka.IsGlobalPoint=False; Kuka.PointName=P59; Kuka.BlendingEnabled=TRUE; Kuka.MoveDataName=CPDATP59; Kuka.VelocityPath=0.068; Kuka.CurrentCDSetIndex=0; Kuka.MovementParameterFieldEnabled=True; IlfCommand=LIN
;ENDFOLD
$BWDSTART = FALSE
LDAT_ACT=LCPDATP59
FDAT_ACT=FP59
BAS (#CP_PARAMS,0.068)
SET_CD_PARAMS (0)
LIN XP59 C_DIS

;ENDFOLD
;FOLD LIN P60 CONT Vel=0.068 m/s CPDATP60 Tool[2] Base[10] ;%{PE}
;FOLD Parameters ;%{h}
;Params IlfProvider=kukaroboter.basistech.inlineforms.movement.old; Kuka.IsGlobalPoint=False; Kuka.PointName=P60; Kuka.BlendingEnabled=TRUE; Kuka.MoveDataName=CPDATP60; Kuka.VelocityPath=0.068; Kuka.CurrentCDSetIndex=0; Kuka.MovementParameterFieldEnabled=True; IlfCommand=LIN
;ENDFOLD
$BWDSTART = FALSE
LDAT_ACT=LCPDATP60
FDAT_ACT=FP60
BAS (#CP_PARAMS,0.068)
SET_CD_PARAMS (0)
LIN XP60 C_DIS

;ENDFOLD
;FOLD LIN P61 CONT Vel=0.068 m/s CPDATP61 Tool[2] Base[10] ;%{PE}
;FOLD Parameters ;%{h}
;Params IlfProvider=kukaroboter.basistech.inlineforms.movement.old; Kuka.IsGlobalPoint=False; Kuka.PointName=P61; Kuka.BlendingEnabled=TRUE; Kuka.MoveDataName=CPDATP61; Kuka.VelocityPath=0.068; Kuka.CurrentCDSetIndex=0; Kuka.MovementParameterFieldEnabled=True; IlfCommand=LIN
;ENDFOLD
$BWDSTART = FALSE
LDAT_ACT=LCPDATP61
FDAT_ACT=FP61
BAS (#CP_PARAMS,0.068)
SET_CD_PARAMS (0)
LIN XP61 C_DIS

;ENDFOLD
;FOLD LIN P62 CONT Vel=0.115 m/s CPDATP62 Tool[2] Base[10] ;%{PE}
;FOLD Parameters ;%{h}
;Params IlfProvider=kukaroboter.basistech.inlineforms.movement.old; Kuka.IsGlobalPoint=False; Kuka.PointName=P62; Kuka.BlendingEnabled=TRUE; Kuka.MoveDataName=CPDATP62; Kuka.VelocityPath=0.115; Kuka.CurrentCDSetIndex=0; Kuka.MovementParameterFieldEnabled=True; IlfCommand=LIN
;ENDFOLD
$BWDSTART = FALSE
LDAT_ACT=LCPDATP62
FDAT_ACT=FP62
BAS (#CP_PARAMS,0.115)
SET_CD_PARAMS (0)
LIN XP62 C_DIS

;ENDFOLD
;FOLD LIN P63 CONT Vel=0.115 m/s CPDATP63 Tool[2] Base[10] ;%{PE}
;FOLD Parameters ;%{h}
;Params IlfProvider=kukaroboter.basistech.inlineforms.movement.old; Kuka.IsGlobalPoint=False; Kuka.PointName=P63; Kuka.BlendingEnabled=TRUE; Kuka.MoveDataName=CPDATP63; Kuka.VelocityPath=0.115; Kuka.CurrentCDSetIndex=0; Kuka.MovementParameterFieldEnabled=True; IlfCommand=LIN
;ENDFOLD
$BWDSTART = FALSE
LDAT_ACT=LCPDATP63
FDAT_ACT=FP63
BAS (#CP_PARAMS,0.115)
SET_CD_PARAMS (0)
LIN XP63 C_DIS

;ENDFOLD
;FOLD LIN P64 CONT Vel=0.115 m/s CPDATP64 Tool[2] Base[10] ;%{PE}
;FOLD Parameters ;%{h}
;Params IlfProvider=kukaroboter.basistech.inlineforms.movement.old; Kuka.IsGlobalPoint=False; Kuka.PointName=P64; Kuka.BlendingEnabled=TRUE; Kuka.MoveDataName=CPDATP64; Kuka.VelocityPath=0.115; Kuka.CurrentCDSetIndex=0; Kuka.MovementParameterFieldEnabled=True; IlfCommand=LIN
;ENDFOLD
$BWDSTART = FALSE
LDAT_ACT=LCPDATP64
FDAT_ACT=FP64
BAS (#CP_PARAMS,0.115)
SET_CD_PARAMS (0)
LIN XP64 C_DIS

;ENDFOLD
;FOLD LIN P65 CONT Vel=0.115 m/s CPDATP65 Tool[2] Base[10] ;%{PE}
;FOLD Parameters ;%{h}
;Params IlfProvider=kukaroboter.basistech.inlineforms.movement.old; Kuka.IsGlobalPoint=False; Kuka.PointName=P65; Kuka.BlendingEnabled=TRUE; Kuka.MoveDataName=CPDATP65; Kuka.VelocityPath=0.115; Kuka.CurrentCDSetIndex=0; Kuka.MovementParameterFieldEnabled=True; IlfCommand=LIN
;ENDFOLD
$BWDSTART = FALSE
LDAT_ACT=LCPDATP65
FDAT_ACT=FP65
BAS (#CP_PARAMS,0.115)
SET_CD_PARAMS (0)
LIN XP65 C_DIS

;ENDFOLD
;FOLD LIN P66 CONT Vel=0.111 m/s CPDATP66 Tool[2] Base[10] ;%{PE}
;FOLD Parameters ;%{h}
;Params IlfProvider=kukaroboter.basistech.inlineforms.movement.old; Kuka.IsGlobalPoint=False; Kuka.PointName=P66; Kuka.BlendingEnabled=TRUE; Kuka.MoveDataName=CPDATP66; Kuka.VelocityPath=0.111; Kuka.CurrentCDSetIndex=0; Kuka.MovementParameterFieldEnabled=True; IlfCommand=LIN
;ENDFOLD
$BWDSTART = FALSE
LDAT_ACT=LCPDATP66
FDAT_ACT=FP66
BAS (#CP_PARAMS,0.111)
SET_CD_PARAMS (0)
LIN XP66 C_DIS

;ENDFOLD
;FOLD LIN P67 CONT Vel=0.111 m/s CPDATP67 Tool[2] Base[10] ;%{PE}
;FOLD Parameters ;%{h}
;Params IlfProvider=kukaroboter.basistech.inlineforms.movement.old; Kuka.IsGlobalPoint=False; Kuka.PointName=P67; Kuka.BlendingEnabled=TRUE; Kuka.MoveDataName=CPDATP67; Kuka.VelocityPath=0.111; Kuka.CurrentCDSetIndex=0; Kuka.MovementParameterFieldEnabled=True; IlfCommand=LIN
;ENDFOLD
$BWDSTART = FALSE
LDAT_ACT=LCPDATP67
FDAT_ACT=FP67
BAS (#CP_PARAMS,0.111)
SET_CD_PARAMS (0)
LIN XP67 C_DIS

;ENDFOLD
;FOLD LIN P68 CONT Vel=0.111 m/s CPDATP68 Tool[2] Base[10] ;%{PE}
;FOLD Parameters ;%{h}
;Params IlfProvider=kukaroboter.basistech.inlineforms.movement.old; Kuka.IsGlobalPoint=False; Kuka.PointName=P68; Kuka.BlendingEnabled=TRUE; Kuka.MoveDataName=CPDATP68; Kuka.VelocityPath=0.111; Kuka.CurrentCDSetIndex=0; Kuka.MovementParameterFieldEnabled=True; IlfCommand=LIN
;ENDFOLD
$BWDSTART = FALSE
LDAT_ACT=LCPDATP68
FDAT_ACT=FP68
BAS (#CP_PARAMS,0.111)
SET_CD_PARAMS (0)
LIN XP68 C_DIS

;ENDFOLD
;FOLD LIN P69 CONT Vel=0.111 m/s CPDATP69 Tool[2] Base[10] ;%{PE}
;FOLD Parameters ;%{h}
;Params IlfProvider=kukaroboter.basistech.inlineforms.movement.old; Kuka.IsGlobalPoint=False; Kuka.PointName=P69; Kuka.BlendingEnabled=TRUE; Kuka.MoveDataName=CPDATP69; Kuka.VelocityPath=0.111; Kuka.CurrentCDSetIndex=0; Kuka.MovementParameterFieldEnabled=True; IlfCommand=LIN
;ENDFOLD
$BWDSTART = FALSE
LDAT_ACT=LCPDATP69
FDAT_ACT=FP69
BAS (#CP_PARAMS,0.111)
SET_CD_PARAMS (0)
LIN XP69 C_DIS

;ENDFOLD
;FOLD LIN P70 CONT Vel=0.124 m/s CPDATP70 Tool[2] Base[10] ;%{PE}
;FOLD Parameters ;%{h}
;Params IlfProvider=kukaroboter.basistech.inlineforms.movement.old; Kuka.IsGlobalPoint=False; Kuka.PointName=P70; Kuka.BlendingEnabled=TRUE; Kuka.MoveDataName=CPDATP70; Kuka.VelocityPath=0.124; Kuka.CurrentCDSetIndex=0; Kuka.MovementParameterFieldEnabled=True; IlfCommand=LIN
;ENDFOLD
$BWDSTART = FALSE
LDAT_ACT=LCPDATP70
FDAT_ACT=FP70
BAS (#CP_PARAMS,0.124)
SET_CD_PARAMS (0)
LIN XP70 C_DIS

;ENDFOLD
;FOLD LIN P71 CONT Vel=0.124 m/s CPDATP71 Tool[2] Base[10] ;%{PE}
;FOLD Parameters ;%{h}
;Params IlfProvider=kukaroboter.basistech.inlineforms.movement.old; Kuka.IsGlobalPoint=False; Kuka.PointName=P71; Kuka.BlendingEnabled=TRUE; Kuka.MoveDataName=CPDATP71; Kuka.VelocityPath=0.124; Kuka.CurrentCDSetIndex=0; Kuka.MovementParameterFieldEnabled=True; IlfCommand=LIN
;ENDFOLD
$BWDSTART = FALSE
LDAT_ACT=LCPDATP71
FDAT_ACT=FP71
BAS (#CP_PARAMS,0.124)
SET_CD_PARAMS (0)
LIN XP71 C_DIS

;ENDFOLD
;FOLD LIN P72 CONT Vel=0.124 m/s CPDATP72 Tool[2] Base[10] ;%{PE}
;FOLD Parameters ;%{h}
;Params IlfProvider=kukaroboter.basistech.inlineforms.movement.old; Kuka.IsGlobalPoint=False; Kuka.PointName=P72; Kuka.BlendingEnabled=TRUE; Kuka.MoveDataName=CPDATP72; Kuka.VelocityPath=0.124; Kuka.CurrentCDSetIndex=0; Kuka.MovementParameterFieldEnabled=True; IlfCommand=LIN
;ENDFOLD
$BWDSTART = FALSE
LDAT_ACT=LCPDATP72
FDAT_ACT=FP72
BAS (#CP_PARAMS,0.124)
SET_CD_PARAMS (0)
LIN XP72 C_DIS

;ENDFOLD
;FOLD LIN P73 CONT Vel=0.124 m/s CPDATP73 Tool[2] Base[10] ;%{PE}
;FOLD Parameters ;%{h}
;Params IlfProvider=kukaroboter.basistech.inlineforms.movement.old; Kuka.IsGlobalPoint=False; Kuka.PointName=P73; Kuka.BlendingEnabled=TRUE; Kuka.MoveDataName=CPDATP73; Kuka.VelocityPath=0.124; Kuka.CurrentCDSetIndex=0; Kuka.MovementParameterFieldEnabled=True; IlfCommand=LIN
;ENDFOLD
$BWDSTART = FALSE
LDAT_ACT=LCPDATP73
FDAT_ACT=FP73
BAS (#CP_PARAMS,0.124)
SET_CD_PARAMS (0)
LIN XP73 C_DIS

;ENDFOLD
;FOLD LIN P74 CONT Vel=0.112 m/s CPDATP74 Tool[2] Base[10] ;%{PE}
;FOLD Parameters ;%{h}
;Params IlfProvider=kukaroboter.basistech.inlineforms.movement.old; Kuka.IsGlobalPoint=False; Kuka.PointName=P74; Kuka.BlendingEnabled=TRUE; Kuka.MoveDataName=CPDATP74; Kuka.VelocityPath=0.112; Kuka.CurrentCDSetIndex=0; Kuka.MovementParameterFieldEnabled=True; IlfCommand=LIN
;ENDFOLD
$BWDSTART = FALSE
LDAT_ACT=LCPDATP74
FDAT_ACT=FP74
BAS (#CP_PARAMS,0.112)
SET_CD_PARAMS (0)
LIN XP74 C_DIS

;ENDFOLD
;FOLD LIN P75 CONT Vel=0.112 m/s CPDATP75 Tool[2] Base[10] ;%{PE}
;FOLD Parameters ;%{h}
;Params IlfProvider=kukaroboter.basistech.inlineforms.movement.old; Kuka.IsGlobalPoint=False; Kuka.PointName=P75; Kuka.BlendingEnabled=TRUE; Kuka.MoveDataName=CPDATP75; Kuka.VelocityPath=0.112; Kuka.CurrentCDSetIndex=0; Kuka.MovementParameterFieldEnabled=True; IlfCommand=LIN
;ENDFOLD
$BWDSTART = FALSE
LDAT_ACT=LCPDATP75
FDAT_ACT=FP75
BAS (#CP_PARAMS,0.112)
SET_CD_PARAMS (0)
LIN XP75 C_DIS

;ENDFOLD
;FOLD LIN P76 CONT Vel=0.112 m/s CPDATP76 Tool[2] Base[10] ;%{PE}
;FOLD Parameters ;%{h}
;Params IlfProvider=kukaroboter.basistech.inlineforms.movement.old; Kuka.IsGlobalPoint=False; Kuka.PointName=P76; Kuka.BlendingEnabled=TRUE; Kuka.MoveDataName=CPDATP76; Kuka.VelocityPath=0.112; Kuka.CurrentCDSetIndex=0; Kuka.MovementParameterFieldEnabled=True; IlfCommand=LIN
;ENDFOLD
$BWDSTART = FALSE
LDAT_ACT=LCPDATP76
FDAT_ACT=FP76
BAS (#CP_PARAMS,0.112)
SET_CD_PARAMS (0)
LIN XP76 C_DIS

;ENDFOLD
;FOLD LIN P77 CONT Vel=0.112 m/s CPDATP77 Tool[2] Base[10] ;%{PE}
;FOLD Parameters ;%{h}
;Params IlfProvider=kukaroboter.basistech.inlineforms.movement.old; Kuka.IsGlobalPoint=False; Kuka.PointName=P77; Kuka.BlendingEnabled=TRUE; Kuka.MoveDataName=CPDATP77; Kuka.VelocityPath=0.112; Kuka.CurrentCDSetIndex=0; Kuka.MovementParameterFieldEnabled=True; IlfCommand=LIN
;ENDFOLD
$BWDSTART = FALSE
LDAT_ACT=LCPDATP77
FDAT_ACT=FP77
BAS (#CP_PARAMS,0.112)
SET_CD_PARAMS (0)
LIN XP77 C_DIS

;ENDFOLD
;FOLD LIN P78 CONT Vel=0.109 m/s CPDATP78 Tool[2] Base[10] ;%{PE}
;FOLD Parameters ;%{h}
;Params IlfProvider=kukaroboter.basistech.inlineforms.movement.old; Kuka.IsGlobalPoint=False; Kuka.PointName=P78; Kuka.BlendingEnabled=TRUE; Kuka.MoveDataName=CPDATP78; Kuka.VelocityPath=0.109; Kuka.CurrentCDSetIndex=0; Kuka.MovementParameterFieldEnabled=True; IlfCommand=LIN
;ENDFOLD
$BWDSTART = FALSE
LDAT_ACT=LCPDATP78
FDAT_ACT=FP78
BAS (#CP_PARAMS,0.109)
SET_CD_PARAMS (0)
LIN XP78 C_DIS

;ENDFOLD
;FOLD LIN P79 CONT Vel=0.109 m/s CPDATP79 Tool[2] Base[10] ;%{PE}
;FOLD Parameters ;%{h}
;Params IlfProvider=kukaroboter.basistech.inlineforms.movement.old; Kuka.IsGlobalPoint=False; Kuka.PointName=P79; Kuka.BlendingEnabled=TRUE; Kuka.MoveDataName=CPDATP79; Kuka.VelocityPath=0.109; Kuka.CurrentCDSetIndex=0; Kuka.MovementParameterFieldEnabled=True; IlfCommand=LIN
;ENDFOLD
$BWDSTART = FALSE
LDAT_ACT=LCPDATP79
FDAT_ACT=FP79
BAS (#CP_PARAMS,0.109)
SET_CD_PARAMS (0)
LIN XP79 C_DIS

;ENDFOLD
;FOLD LIN P80 CONT Vel=0.109 m/s CPDATP80 Tool[2] Base[10] ;%{PE}
;FOLD Parameters ;%{h}
;Params IlfProvider=kukaroboter.basistech.inlineforms.movement.old; Kuka.IsGlobalPoint=False; Kuka.PointName=P80; Kuka.BlendingEnabled=TRUE; Kuka.MoveDataName=CPDATP80; Kuka.VelocityPath=0.109; Kuka.CurrentCDSetIndex=0; Kuka.MovementParameterFieldEnabled=True; IlfCommand=LIN
;ENDFOLD
$BWDSTART = FALSE
LDAT_ACT=LCPDATP80
FDAT_ACT=FP80
BAS (#CP_PARAMS,0.109)
SET_CD_PARAMS (0)
LIN XP80 C_DIS

;ENDFOLD
;FOLD LIN P81 CONT Vel=0.109 m/s CPDATP81 Tool[2] Base[10] ;%{PE}
;FOLD Parameters ;%{h}
;Params IlfProvider=kukaroboter.basistech.inlineforms.movement.old; Kuka.IsGlobalPoint=False; Kuka.PointName=P81; Kuka.BlendingEnabled=TRUE; Kuka.MoveDataName=CPDATP81; Kuka.VelocityPath=0.109; Kuka.CurrentCDSetIndex=0; Kuka.MovementParameterFieldEnabled=True; IlfCommand=LIN
;ENDFOLD
$BWDSTART = FALSE
LDAT_ACT=LCPDATP81
FDAT_ACT=FP81
BAS (#CP_PARAMS,0.109)
SET_CD_PARAMS (0)
LIN XP81 C_DIS

;ENDFOLD
;FOLD LIN P82 CONT Vel=0.104 m/s CPDATP82 Tool[2] Base[10] ;%{PE}
;FOLD Parameters ;%{h}
;Params IlfProvider=kukaroboter.basistech.inlineforms.movement.old; Kuka.IsGlobalPoint=False; Kuka.PointName=P82; Kuka.BlendingEnabled=TRUE; Kuka.MoveDataName=CPDATP82; Kuka.VelocityPath=0.104; Kuka.CurrentCDSetIndex=0; Kuka.MovementParameterFieldEnabled=True; IlfCommand=LIN
;ENDFOLD
$BWDSTART = FALSE
LDAT_ACT=LCPDATP82
FDAT_ACT=FP82
BAS (#CP_PARAMS,0.104)
SET_CD_PARAMS (0)
LIN XP82 C_DIS

;ENDFOLD
;FOLD LIN P83 CONT Vel=0.104 m/s CPDATP83 Tool[2] Base[10] ;%{PE}
;FOLD Parameters ;%{h}
;Params IlfProvider=kukaroboter.basistech.inlineforms.movement.old; Kuka.IsGlobalPoint=False; Kuka.PointName=P83; Kuka.BlendingEnabled=TRUE; Kuka.MoveDataName=CPDATP83; Kuka.VelocityPath=0.104; Kuka.CurrentCDSetIndex=0; Kuka.MovementParameterFieldEnabled=True; IlfCommand=LIN
;ENDFOLD
$BWDSTART = FALSE
LDAT_ACT=LCPDATP83
FDAT_ACT=FP83
BAS (#CP_PARAMS,0.104)
SET_CD_PARAMS (0)
LIN XP83 C_DIS

;ENDFOLD
;FOLD LIN P84 CONT Vel=0.104 m/s CPDATP84 Tool[2] Base[10] ;%{PE}
;FOLD Parameters ;%{h}
;Params IlfProvider=kukaroboter.basistech.inlineforms.movement.old; Kuka.IsGlobalPoint=False; Kuka.PointName=P84; Kuka.BlendingEnabled=TRUE; Kuka.MoveDataName=CPDATP84; Kuka.VelocityPath=0.104; Kuka.CurrentCDSetIndex=0; Kuka.MovementParameterFieldEnabled=True; IlfCommand=LIN
;ENDFOLD
$BWDSTART = FALSE
LDAT_ACT=LCPDATP84
FDAT_ACT=FP84
BAS (#CP_PARAMS,0.104)
SET_CD_PARAMS (0)
LIN XP84 C_DIS

;ENDFOLD
;FOLD LIN P85 CONT Vel=0.104 m/s CPDATP85 Tool[2] Base[10] ;%{PE}
;FOLD Parameters ;%{h}
;Params IlfProvider=kukaroboter.basistech.inlineforms.movement.old; Kuka.IsGlobalPoint=False; Kuka.PointName=P85; Kuka.BlendingEnabled=TRUE; Kuka.MoveDataName=CPDATP85; Kuka.VelocityPath=0.104; Kuka.CurrentCDSetIndex=0; Kuka.MovementParameterFieldEnabled=True; IlfCommand=LIN
;ENDFOLD
$BWDSTART = FALSE
LDAT_ACT=LCPDATP85
FDAT_ACT=FP85
BAS (#CP_PARAMS,0.104)
SET_CD_PARAMS (0)
LIN XP85 C_DIS

;ENDFOLD
;FOLD LIN P86 CONT Vel=0.053 m/s CPDATP86 Tool[2] Base[10] ;%{PE}
;FOLD Parameters ;%{h}
;Params IlfProvider=kukaroboter.basistech.inlineforms.movement.old; Kuka.IsGlobalPoint=False; Kuka.PointName=P86; Kuka.BlendingEnabled=TRUE; Kuka.MoveDataName=CPDATP86; Kuka.VelocityPath=0.053; Kuka.CurrentCDSetIndex=0; Kuka.MovementParameterFieldEnabled=True; IlfCommand=LIN
;ENDFOLD
$BWDSTART = FALSE
LDAT_ACT=LCPDATP86
FDAT_ACT=FP86
BAS (#CP_PARAMS,0.053)
SET_CD_PARAMS (0)
LIN XP86 C_DIS

;ENDFOLD
;FOLD LIN P87 CONT Vel=0.053 m/s CPDATP87 Tool[2] Base[10] ;%{PE}
;FOLD Parameters ;%{h}
;Params IlfProvider=kukaroboter.basistech.inlineforms.movement.old; Kuka.IsGlobalPoint=False; Kuka.PointName=P87; Kuka.BlendingEnabled=TRUE; Kuka.MoveDataName=CPDATP87; Kuka.VelocityPath=0.053; Kuka.CurrentCDSetIndex=0; Kuka.MovementParameterFieldEnabled=True; IlfCommand=LIN
;ENDFOLD
$BWDSTART = FALSE
LDAT_ACT=LCPDATP87
FDAT_ACT=FP87
BAS (#CP_PARAMS,0.053)
SET_CD_PARAMS (0)
LIN XP87 C_DIS

;ENDFOLD
;FOLD LIN P88 CONT Vel=0.053 m/s CPDATP88 Tool[2] Base[10] ;%{PE}
;FOLD Parameters ;%{h}
;Params IlfProvider=kukaroboter.basistech.inlineforms.movement.old; Kuka.IsGlobalPoint=False; Kuka.PointName=P88; Kuka.BlendingEnabled=TRUE; Kuka.MoveDataName=CPDATP88; Kuka.VelocityPath=0.053; Kuka.CurrentCDSetIndex=0; Kuka.MovementParameterFieldEnabled=True; IlfCommand=LIN
;ENDFOLD
$BWDSTART = FALSE
LDAT_ACT=LCPDATP88
FDAT_ACT=FP88
BAS (#CP_PARAMS,0.053)
SET_CD_PARAMS (0)
LIN XP88 C_DIS

;ENDFOLD
;FOLD LIN P89 CONT Vel=0.053 m/s CPDATP89 Tool[2] Base[10] ;%{PE}
;FOLD Parameters ;%{h}
;Params IlfProvider=kukaroboter.basistech.inlineforms.movement.old; Kuka.IsGlobalPoint=False; Kuka.PointName=P89; Kuka.BlendingEnabled=TRUE; Kuka.MoveDataName=CPDATP89; Kuka.VelocityPath=0.053; Kuka.CurrentCDSetIndex=0; Kuka.MovementParameterFieldEnabled=True; IlfCommand=LIN
;ENDFOLD
$BWDSTART = FALSE
LDAT_ACT=LCPDATP89
FDAT_ACT=FP89
BAS (#CP_PARAMS,0.053)
SET_CD_PARAMS (0)
LIN XP89 C_DIS

;ENDFOLD
;FOLD LIN P90 CONT Vel=0.063 m/s CPDATP90 Tool[2] Base[10] ;%{PE}
;FOLD Parameters ;%{h}
;Params IlfProvider=kukaroboter.basistech.inlineforms.movement.old; Kuka.IsGlobalPoint=False; Kuka.PointName=P90; Kuka.BlendingEnabled=TRUE; Kuka.MoveDataName=CPDATP90; Kuka.VelocityPath=0.063; Kuka.CurrentCDSetIndex=0; Kuka.MovementParameterFieldEnabled=True; IlfCommand=LIN
;ENDFOLD
$BWDSTART = FALSE
LDAT_ACT=LCPDATP90
FDAT_ACT=FP90
BAS (#CP_PARAMS,0.063)
SET_CD_PARAMS (0)
LIN XP90 C_DIS

;ENDFOLD
;FOLD LIN P91 CONT Vel=0.063 m/s CPDATP91 Tool[2] Base[10] ;%{PE}
;FOLD Parameters ;%{h}
;Params IlfProvider=kukaroboter.basistech.inlineforms.movement.old; Kuka.IsGlobalPoint=False; Kuka.PointName=P91; Kuka.BlendingEnabled=TRUE; Kuka.MoveDataName=CPDATP91; Kuka.VelocityPath=0.063; Kuka.CurrentCDSetIndex=0; Kuka.MovementParameterFieldEnabled=True; IlfCommand=LIN
;ENDFOLD
$BWDSTART = FALSE
LDAT_ACT=LCPDATP91
FDAT_ACT=FP91
BAS (#CP_PARAMS,0.063)
SET_CD_PARAMS (0)
LIN XP91 C_DIS

;ENDFOLD
;FOLD LIN P92 CONT Vel=0.063 m/s CPDATP92 Tool[2] Base[10] ;%{PE}
;FOLD Parameters ;%{h}
;Params IlfProvider=kukaroboter.basistech.inlineforms.movement.old; Kuka.IsGlobalPoint=False; Kuka.PointName=P92; Kuka.BlendingEnabled=TRUE; Kuka.MoveDataName=CPDATP92; Kuka.VelocityPath=0.063; Kuka.CurrentCDSetIndex=0; Kuka.MovementParameterFieldEnabled=True; IlfCommand=LIN
;ENDFOLD
$BWDSTART = FALSE
LDAT_ACT=LCPDATP92
FDAT_ACT=FP92
BAS (#CP_PARAMS,0.063)
SET_CD_PARAMS (0)
LIN XP92 C_DIS

;ENDFOLD
;FOLD LIN P93 CONT Vel=0.063 m/s CPDATP93 Tool[2] Base[10] ;%{PE}
;FOLD Parameters ;%{h}
;Params IlfProvider=kukaroboter.basistech.inlineforms.movement.old; Kuka.IsGlobalPoint=False; Kuka.PointName=P93; Kuka.BlendingEnabled=TRUE; Kuka.MoveDataName=CPDATP93; Kuka.VelocityPath=0.063; Kuka.CurrentCDSetIndex=0; Kuka.MovementParameterFieldEnabled=True; IlfCommand=LIN
;ENDFOLD
$BWDSTART = FALSE
LDAT_ACT=LCPDATP93
FDAT_ACT=FP93
BAS (#CP_PARAMS,0.063)
SET_CD_PARAMS (0)
LIN XP93 C_DIS

;ENDFOLD
;FOLD LIN P94 CONT Vel=0.5 m/s CPDATP94 Tool[2] Base[10] ;%{PE}
;FOLD Parameters ;%{h}
;Params IlfProvider=kukaroboter.basistech.inlineforms.movement.old; Kuka.IsGlobalPoint=False; Kuka.PointName=P94; Kuka.BlendingEnabled=TRUE; Kuka.MoveDataName=CPDATP94; Kuka.VelocityPath=0.5; Kuka.CurrentCDSetIndex=0; Kuka.MovementParameterFieldEnabled=True; IlfCommand=LIN
;ENDFOLD
$BWDSTART = FALSE
LDAT_ACT=LCPDATP94
FDAT_ACT=FP94
BAS (#CP_PARAMS,0.5)
SET_CD_PARAMS (0)
LIN XP94 C_DIS

;ENDFOLD
;FOLD LIN P95 CONT Vel=1.0 m/s CPDATP95 Tool[2] Base[10] ;%{PE}
;FOLD Parameters ;%{h}
;Params IlfProvider=kukaroboter.basistech.inlineforms.movement.old; Kuka.IsGlobalPoint=False; Kuka.PointName=P95; Kuka.BlendingEnabled=TRUE; Kuka.MoveDataName=CPDATP95; Kuka.VelocityPath=1.0; Kuka.CurrentCDSetIndex=0; Kuka.MovementParameterFieldEnabled=True; IlfCommand=LIN
;ENDFOLD
$BWDSTART = FALSE
LDAT_ACT=LCPDATP95
FDAT_ACT=FP95
BAS (#CP_PARAMS,1.0)
SET_CD_PARAMS (0)
LIN XP95 C_DIS

;ENDFOLD
;FOLD LIN P96 CONT Vel=1.0 m/s CPDATP96 Tool[2] Base[10] ;%{PE}
;FOLD Parameters ;%{h}
;Params IlfProvider=kukaroboter.basistech.inlineforms.movement.old; Kuka.IsGlobalPoint=False; Kuka.PointName=P96; Kuka.BlendingEnabled=TRUE; Kuka.MoveDataName=CPDATP96; Kuka.VelocityPath=1.0; Kuka.CurrentCDSetIndex=0; Kuka.MovementParameterFieldEnabled=True; IlfCommand=LIN
;ENDFOLD
$BWDSTART = FALSE
LDAT_ACT=LCPDATP96
FDAT_ACT=FP96
BAS (#CP_PARAMS,1.0)
SET_CD_PARAMS (0)
LIN XP96 C_DIS

;ENDFOLD
END
;End of routine {i}

; --- Routine for substrate 1 ---
DEF Routine_1()
;FOLD LIN P97 CONT Vel=1.0 m/s CPDATP97 Tool[2] Base[9] ;%{PE}
;FOLD Parameters ;%{h}
;Params IlfProvider=kukaroboter.basistech.inlineforms.movement.old; Kuka.IsGlobalPoint=False; Kuka.PointName=P97; Kuka.BlendingEnabled=TRUE; Kuka.MoveDataName=CPDATP97; Kuka.VelocityPath=1.0; Kuka.CurrentCDSetIndex=0; Kuka.MovementParameterFieldEnabled=True; IlfCommand=LIN
;ENDFOLD
$BWDSTART = FALSE
LDAT_ACT=LCPDATP97
FDAT_ACT=FP97
BAS (#CP_PARAMS,1.0)
SET_CD_PARAMS (0)
LIN XP97 C_DIS

;ENDFOLD
;FOLD LIN P98 CONT Vel=0.065 m/s CPDATP98 Tool[2] Base[9] ;%{PE}
;FOLD Parameters ;%{h}
;Params IlfProvider=kukaroboter.basistech.inlineforms.movement.old; Kuka.IsGlobalPoint=False; Kuka.PointName=P98; Kuka.BlendingEnabled=TRUE; Kuka.MoveDataName=CPDATP98; Kuka.VelocityPath=0.065; Kuka.CurrentCDSetIndex=0; Kuka.MovementParameterFieldEnabled=True; IlfCommand=LIN
;ENDFOLD
$BWDSTART = FALSE
LDAT_ACT=LCPDATP98
FDAT_ACT=FP98
BAS (#CP_PARAMS,0.065)
SET_CD_PARAMS (0)
LIN XP98 C_DIS

;ENDFOLD
;FOLD LIN P99 CONT Vel=0.065 m/s CPDATP99 Tool[2] Base[9] ;%{PE}
;FOLD Parameters ;%{h}
;Params IlfProvider=kukaroboter.basistech.inlineforms.movement.old; Kuka.IsGlobalPoint=False; Kuka.PointName=P99; Kuka.BlendingEnabled=TRUE; Kuka.MoveDataName=CPDATP99; Kuka.VelocityPath=0.065; Kuka.CurrentCDSetIndex=0; Kuka.MovementParameterFieldEnabled=True; IlfCommand=LIN
;ENDFOLD
$BWDSTART = FALSE
LDAT_ACT=LCPDATP99
FDAT_ACT=FP99
BAS (#CP_PARAMS,0.065)
SET_CD_PARAMS (0)
LIN XP99 C_DIS

;ENDFOLD
;FOLD LIN P100 CONT Vel=0.065 m/s CPDATP100 Tool[2] Base[9] ;%{PE}
;FOLD Parameters ;%{h}
;Params IlfProvider=kukaroboter.basistech.inlineforms.movement.old; Kuka.IsGlobalPoint=False; Kuka.PointName=P100; Kuka.BlendingEnabled=TRUE; Kuka.MoveDataName=CPDATP100; Kuka.VelocityPath=0.065; Kuka.CurrentCDSetIndex=0; Kuka.MovementParameterFieldEnabled=True; IlfCommand=LIN
;ENDFOLD
$BWDSTART = FALSE
LDAT_ACT=LCPDATP100
FDAT_ACT=FP100
BAS (#CP_PARAMS,0.065)
SET_CD_PARAMS (0)
LIN XP100 C_DIS

;ENDFOLD
;FOLD LIN P101 CONT Vel=0.065 m/s CPDATP101 Tool[2] Base[9] ;%{PE}
;FOLD Parameters ;%{h}
;Params IlfProvider=kukaroboter.basistech.inlineforms.movement.old; Kuka.IsGlobalPoint=False; Kuka.PointName=P101; Kuka.BlendingEnabled=TRUE; Kuka.MoveDataName=CPDATP101; Kuka.VelocityPath=0.065; Kuka.CurrentCDSetIndex=0; Kuka.MovementParameterFieldEnabled=True; IlfCommand=LIN
;ENDFOLD
$BWDSTART = FALSE
LDAT_ACT=LCPDATP101
FDAT_ACT=FP101
BAS (#CP_PARAMS,0.065)
SET_CD_PARAMS (0)
LIN XP101 C_DIS

;ENDFOLD
;FOLD LIN P102 CONT Vel=0.088 m/s CPDATP102 Tool[2] Base[9] ;%{PE}
;FOLD Parameters ;%{h}
;Params IlfProvider=kukaroboter.basistech.inlineforms.movement.old; Kuka.IsGlobalPoint=False; Kuka.PointName=P102; Kuka.BlendingEnabled=TRUE; Kuka.MoveDataName=CPDATP102; Kuka.VelocityPath=0.088; Kuka.CurrentCDSetIndex=0; Kuka.MovementParameterFieldEnabled=True; IlfCommand=LIN
;ENDFOLD
$BWDSTART = FALSE
LDAT_ACT=LCPDATP102
FDAT_ACT=FP102
BAS (#CP_PARAMS,0.088)
SET_CD_PARAMS (0)
LIN XP102 C_DIS

;ENDFOLD
;FOLD LIN P103 CONT Vel=0.088 m/s CPDATP103 Tool[2] Base[9] ;%{PE}
;FOLD Parameters ;%{h}
;Params IlfProvider=kukaroboter.basistech.inlineforms.movement.old; Kuka.IsGlobalPoint=False; Kuka.PointName=P103; Kuka.BlendingEnabled=TRUE; Kuka.MoveDataName=CPDATP103; Kuka.VelocityPath=0.088; Kuka.CurrentCDSetIndex=0; Kuka.MovementParameterFieldEnabled=True; IlfCommand=LIN
;ENDFOLD
$BWDSTART = FALSE
LDAT_ACT=LCPDATP103
FDAT_ACT=FP103
BAS (#CP_PARAMS,0.088)
SET_CD_PARAMS (0)
LIN XP103 C_DIS

;ENDFOLD
;FOLD LIN P104 CONT Vel=0.088 m/s CPDATP104 Tool[2] Base[9] ;%{PE}
;FOLD Parameters ;%{h}
;Params IlfProvider=kukaroboter.basistech.inlineforms.movement.old; Kuka.IsGlobalPoint=False; Kuka.PointName=P104; Kuka.BlendingEnabled=TRUE; Kuka.MoveDataName=CPDATP104; Kuka.VelocityPath=0.088; Kuka.CurrentCDSetIndex=0; Kuka.MovementParameterFieldEnabled=True; IlfCommand=LIN
;ENDFOLD
$BWDSTART = FALSE
LDAT_ACT=LCPDATP104
FDAT_ACT=FP104
BAS (#CP_PARAMS,0.088)
SET_CD_PARAMS (0)
LIN XP104 C_DIS

;ENDFOLD
;FOLD LIN P105 CONT Vel=0.088 m/s CPDATP105 Tool[2] Base[9] ;%{PE}
;FOLD Parameters ;%{h}
;Params IlfProvider=kukaroboter.basistech.inlineforms.movement.old; Kuka.IsGlobalPoint=False; Kuka.PointName=P105; Kuka.BlendingEnabled=TRUE; Kuka.MoveDataName=CPDATP105; Kuka.VelocityPath=0.088; Kuka.CurrentCDSetIndex=0; Kuka.MovementParameterFieldEnabled=True; IlfCommand=LIN
;ENDFOLD
$BWDSTART = FALSE
LDAT_ACT=LCPDATP105
FDAT_ACT=FP105
BAS (#CP_PARAMS,0.088)
SET_CD_PARAMS (0)
LIN XP105 C_DIS

;ENDFOLD
;FOLD LIN P106 CONT Vel=0.06 m/s CPDATP106 Tool[2] Base[9] ;%{PE}
;FOLD Parameters ;%{h}
;Params IlfProvider=kukaroboter.basistech.inlineforms.movement.old; Kuka.IsGlobalPoint=False; Kuka.PointName=P106; Kuka.BlendingEnabled=TRUE; Kuka.MoveDataName=CPDATP106; Kuka.VelocityPath=0.06; Kuka.CurrentCDSetIndex=0; Kuka.MovementParameterFieldEnabled=True; IlfCommand=LIN
;ENDFOLD
$BWDSTART = FALSE
LDAT_ACT=LCPDATP106
FDAT_ACT=FP106
BAS (#CP_PARAMS,0.06)
SET_CD_PARAMS (0)
LIN XP106 C_DIS

;ENDFOLD
;FOLD LIN P107 CONT Vel=0.06 m/s CPDATP107 Tool[2] Base[9] ;%{PE}
;FOLD Parameters ;%{h}
;Params IlfProvider=kukaroboter.basistech.inlineforms.movement.old; Kuka.IsGlobalPoint=False; Kuka.PointName=P107; Kuka.BlendingEnabled=TRUE; Kuka.MoveDataName=CPDATP107; Kuka.VelocityPath=0.06; Kuka.CurrentCDSetIndex=0; Kuka.MovementParameterFieldEnabled=True; IlfCommand=LIN
;ENDFOLD
$BWDSTART = FALSE
LDAT_ACT=LCPDATP107
FDAT_ACT=FP107
BAS (#CP_PARAMS,0.06)
SET_CD_PARAMS (0)
LIN XP107 C_DIS

;ENDFOLD
;FOLD LIN P108 CONT Vel=0.06 m/s CPDATP108 Tool[2] Base[9] ;%{PE}
;FOLD Parameters ;%{h}
;Params IlfProvider=kukaroboter.basistech.inlineforms.movement.old; Kuka.IsGlobalPoint=False; Kuka.PointName=P108; Kuka.BlendingEnabled=TRUE; Kuka.MoveDataName=CPDATP108; Kuka.VelocityPath=0.06; Kuka.CurrentCDSetIndex=0; Kuka.MovementParameterFieldEnabled=True; IlfCommand=LIN
;ENDFOLD
$BWDSTART = FALSE
LDAT_ACT=LCPDATP108
FDAT_ACT=FP108
BAS (#CP_PARAMS,0.06)
SET_CD_PARAMS (0)
LIN XP108 C_DIS

;ENDFOLD
;FOLD LIN P109 CONT Vel=0.06 m/s CPDATP109 Tool[2] Base[9] ;%{PE}
;FOLD Parameters ;%{h}
;Params IlfProvider=kukaroboter.basistech.inlineforms.movement.old; Kuka.IsGlobalPoint=False; Kuka.PointName=P109; Kuka.BlendingEnabled=TRUE; Kuka.MoveDataName=CPDATP109; Kuka.VelocityPath=0.06; Kuka.CurrentCDSetIndex=0; Kuka.MovementParameterFieldEnabled=True; IlfCommand=LIN
;ENDFOLD
$BWDSTART = FALSE
LDAT_ACT=LCPDATP109
FDAT_ACT=FP109
BAS (#CP_PARAMS,0.06)
SET_CD_PARAMS (0)
LIN XP109 C_DIS

;ENDFOLD
;FOLD LIN P110 CONT Vel=0.135 m/s CPDATP110 Tool[2] Base[9] ;%{PE}
;FOLD Parameters ;%{h}
;Params IlfProvider=kukaroboter.basistech.inlineforms.movement.old; Kuka.IsGlobalPoint=False; Kuka.PointName=P110; Kuka.BlendingEnabled=TRUE; Kuka.MoveDataName=CPDATP110; Kuka.VelocityPath=0.135; Kuka.CurrentCDSetIndex=0; Kuka.MovementParameterFieldEnabled=True; IlfCommand=LIN
;ENDFOLD
$BWDSTART = FALSE
LDAT_ACT=LCPDATP110
FDAT_ACT=FP110
BAS (#CP_PARAMS,0.135)
SET_CD_PARAMS (0)
LIN XP110 C_DIS

;ENDFOLD
;FOLD LIN P111 CONT Vel=0.135 m/s CPDATP111 Tool[2] Base[9] ;%{PE}
;FOLD Parameters ;%{h}
;Params IlfProvider=kukaroboter.basistech.inlineforms.movement.old; Kuka.IsGlobalPoint=False; Kuka.PointName=P111; Kuka.BlendingEnabled=TRUE; Kuka.MoveDataName=CPDATP111; Kuka.VelocityPath=0.135; Kuka.CurrentCDSetIndex=0; Kuka.MovementParameterFieldEnabled=True; IlfCommand=LIN
;ENDFOLD
$BWDSTART = FALSE
LDAT_ACT=LCPDATP111
FDAT_ACT=FP111
BAS (#CP_PARAMS,0.135)
SET_CD_PARAMS (0)
LIN XP111 C_DIS

;ENDFOLD
;FOLD LIN P112 CONT Vel=0.135 m/s CPDATP112 Tool[2] Base[9] ;%{PE}
;FOLD Parameters ;%{h}
;Params IlfProvider=kukaroboter.basistech.inlineforms.movement.old; Kuka.IsGlobalPoint=False; Kuka.PointName=P112; Kuka.BlendingEnabled=TRUE; Kuka.MoveDataName=CPDATP112; Kuka.VelocityPath=0.135; Kuka.CurrentCDSetIndex=0; Kuka.MovementParameterFieldEnabled=True; IlfCommand=LIN
;ENDFOLD
$BWDSTART = FALSE
LDAT_ACT=LCPDATP112
FDAT_ACT=FP112
BAS (#CP_PARAMS,0.135)
SET_CD_PARAMS (0)
LIN XP112 C_DIS

;ENDFOLD
;FOLD LIN P113 CONT Vel=0.135 m/s CPDATP113 Tool[2] Base[9] ;%{PE}
;FOLD Parameters ;%{h}
;Params IlfProvider=kukaroboter.basistech.inlineforms.movement.old; Kuka.IsGlobalPoint=False; Kuka.PointName=P113; Kuka.BlendingEnabled=TRUE; Kuka.MoveDataName=CPDATP113; Kuka.VelocityPath=0.135; Kuka.CurrentCDSetIndex=0; Kuka.MovementParameterFieldEnabled=True; IlfCommand=LIN
;ENDFOLD
$BWDSTART = FALSE
LDAT_ACT=LCPDATP113
FDAT_ACT=FP113
BAS (#CP_PARAMS,0.135)
SET_CD_PARAMS (0)
LIN XP113 C_DIS

;ENDFOLD
;FOLD LIN P114 CONT Vel=0.119 m/s CPDATP114 Tool[2] Base[9] ;%{PE}
;FOLD Parameters ;%{h}
;Params IlfProvider=kukaroboter.basistech.inlineforms.movement.old; Kuka.IsGlobalPoint=False; Kuka.PointName=P114; Kuka.BlendingEnabled=TRUE; Kuka.MoveDataName=CPDATP114; Kuka.VelocityPath=0.119; Kuka.CurrentCDSetIndex=0; Kuka.MovementParameterFieldEnabled=True; IlfCommand=LIN
;ENDFOLD
$BWDSTART = FALSE
LDAT_ACT=LCPDATP114
FDAT_ACT=FP114
BAS (#CP_PARAMS,0.119)
SET_CD_PARAMS (0)
LIN XP114 C_DIS

;ENDFOLD
;FOLD LIN P115 CONT Vel=0.119 m/s CPDATP115 Tool[2] Base[9] ;%{PE}
;FOLD Parameters ;%{h}
;Params IlfProvider=kukaroboter.basistech.inlineforms.movement.old; Kuka.IsGlobalPoint=False; Kuka.PointName=P115; Kuka.BlendingEnabled=TRUE; Kuka.MoveDataName=CPDATP115; Kuka.VelocityPath=0.119; Kuka.CurrentCDSetIndex=0; Kuka.MovementParameterFieldEnabled=True; IlfCommand=LIN
;ENDFOLD
$BWDSTART = FALSE
LDAT_ACT=LCPDATP115
FDAT_ACT=FP115
BAS (#CP_PARAMS,0.119)
SET_CD_PARAMS (0)
LIN XP115 C_DIS

;ENDFOLD
;FOLD LIN P116 CONT Vel=0.119 m/s CPDATP116 Tool[2] Base[9] ;%{PE}
;FOLD Parameters ;%{h}
;Params IlfProvider=kukaroboter.basistech.inlineforms.movement.old; Kuka.IsGlobalPoint=False; Kuka.PointName=P116; Kuka.BlendingEnabled=TRUE; Kuka.MoveDataName=CPDATP116; Kuka.VelocityPath=0.119; Kuka.CurrentCDSetIndex=0; Kuka.MovementParameterFieldEnabled=True; IlfCommand=LIN
;ENDFOLD
$BWDSTART = FALSE
LDAT_ACT=LCPDATP116
FDAT_ACT=FP116
BAS (#CP_PARAMS,0.119)
SET_CD_PARAMS (0)
LIN XP116 C_DIS

;ENDFOLD
;FOLD LIN P117 CONT Vel=0.119 m/s CPDATP117 Tool[2] Base[9] ;%{PE}
;FOLD Parameters ;%{h}
;Params IlfProvider=kukaroboter.basistech.inlineforms.movement.old; Kuka.IsGlobalPoint=False; Kuka.PointName=P117; Kuka.BlendingEnabled=TRUE; Kuka.MoveDataName=CPDATP117; Kuka.VelocityPath=0.119; Kuka.CurrentCDSetIndex=0; Kuka.MovementParameterFieldEnabled=True; IlfCommand=LIN
;ENDFOLD
$BWDSTART = FALSE
LDAT_ACT=LCPDATP117
FDAT_ACT=FP117
BAS (#CP_PARAMS,0.119)
SET_CD_PARAMS (0)
LIN XP117 C_DIS

;ENDFOLD
;FOLD LIN P118 CONT Vel=0.069 m/s CPDATP118 Tool[2] Base[9] ;%{PE}
;FOLD Parameters ;%{h}
;Params IlfProvider=kukaroboter.basistech.inlineforms.movement.old; Kuka.IsGlobalPoint=False; Kuka.PointName=P118; Kuka.BlendingEnabled=TRUE; Kuka.MoveDataName=CPDATP118; Kuka.VelocityPath=0.069; Kuka.CurrentCDSetIndex=0; Kuka.MovementParameterFieldEnabled=True; IlfCommand=LIN
;ENDFOLD
$BWDSTART = FALSE
LDAT_ACT=LCPDATP118
FDAT_ACT=FP118
BAS (#CP_PARAMS,0.069)
SET_CD_PARAMS (0)
LIN XP118 C_DIS

;ENDFOLD
;FOLD LIN P119 CONT Vel=0.069 m/s CPDATP119 Tool[2] Base[9] ;%{PE}
;FOLD Parameters ;%{h}
;Params IlfProvider=kukaroboter.basistech.inlineforms.movement.old; Kuka.IsGlobalPoint=False; Kuka.PointName=P119; Kuka.BlendingEnabled=TRUE; Kuka.MoveDataName=CPDATP119; Kuka.VelocityPath=0.069; Kuka.CurrentCDSetIndex=0; Kuka.MovementParameterFieldEnabled=True; IlfCommand=LIN
;ENDFOLD
$BWDSTART = FALSE
LDAT_ACT=LCPDATP119
FDAT_ACT=FP119
BAS (#CP_PARAMS,0.069)
SET_CD_PARAMS (0)
LIN XP119 C_DIS

;ENDFOLD
;FOLD LIN P120 CONT Vel=0.069 m/s CPDATP120 Tool[2] Base[9] ;%{PE}
;FOLD Parameters ;%{h}
;Params IlfProvider=kukaroboter.basistech.inlineforms.movement.old; Kuka.IsGlobalPoint=False; Kuka.PointName=P120; Kuka.BlendingEnabled=TRUE; Kuka.MoveDataName=CPDATP120; Kuka.VelocityPath=0.069; Kuka.CurrentCDSetIndex=0; Kuka.MovementParameterFieldEnabled=True; IlfCommand=LIN
;ENDFOLD
$BWDSTART = FALSE
LDAT_ACT=LCPDATP120
FDAT_ACT=FP120
BAS (#CP_PARAMS,0.069)
SET_CD_PARAMS (0)
LIN XP120 C_DIS

;ENDFOLD
;FOLD LIN P121 CONT Vel=0.069 m/s CPDATP121 Tool[2] Base[9] ;%{PE}
;FOLD Parameters ;%{h}
;Params IlfProvider=kukaroboter.basistech.inlineforms.movement.old; Kuka.IsGlobalPoint=False; Kuka.PointName=P121; Kuka.BlendingEnabled=TRUE; Kuka.MoveDataName=CPDATP121; Kuka.VelocityPath=0.069; Kuka.CurrentCDSetIndex=0; Kuka.MovementParameterFieldEnabled=True; IlfCommand=LIN
;ENDFOLD
$BWDSTART = FALSE
LDAT_ACT=LCPDATP121
FDAT_ACT=FP121
BAS (#CP_PARAMS,0.069)
SET_CD_PARAMS (0)
LIN XP121 C_DIS

;ENDFOLD
;FOLD LIN P122 CONT Vel=0.093 m/s CPDATP122 Tool[2] Base[9] ;%{PE}
;FOLD Parameters ;%{h}
;Params IlfProvider=kukaroboter.basistech.inlineforms.movement.old; Kuka.IsGlobalPoint=False; Kuka.PointName=P122; Kuka.BlendingEnabled=TRUE; Kuka.MoveDataName=CPDATP122; Kuka.VelocityPath=0.093; Kuka.CurrentCDSetIndex=0; Kuka.MovementParameterFieldEnabled=True; IlfCommand=LIN
;ENDFOLD
$BWDSTART = FALSE
LDAT_ACT=LCPDATP122
FDAT_ACT=FP122
BAS (#CP_PARAMS,0.093)
SET_CD_PARAMS (0)
LIN XP122 C_DIS

;ENDFOLD
;FOLD LIN P123 CONT Vel=0.093 m/s CPDATP123 Tool[2] Base[9] ;%{PE}
;FOLD Parameters ;%{h}
;Params IlfProvider=kukaroboter.basistech.inlineforms.movement.old; Kuka.IsGlobalPoint=False; Kuka.PointName=P123; Kuka.BlendingEnabled=TRUE; Kuka.MoveDataName=CPDATP123; Kuka.VelocityPath=0.093; Kuka.CurrentCDSetIndex=0; Kuka.MovementParameterFieldEnabled=True; IlfCommand=LIN
;ENDFOLD
$BWDSTART = FALSE
LDAT_ACT=LCPDATP123
FDAT_ACT=FP123
BAS (#CP_PARAMS,0.093)
SET_CD_PARAMS (0)
LIN XP123 C_DIS

;ENDFOLD
;FOLD LIN P124 CONT Vel=0.093 m/s CPDATP124 Tool[2] Base[9] ;%{PE}
;FOLD Parameters ;%{h}
;Params IlfProvider=kukaroboter.basistech.inlineforms.movement.old; Kuka.IsGlobalPoint=False; Kuka.PointName=P124; Kuka.BlendingEnabled=TRUE; Kuka.MoveDataName=CPDATP124; Kuka.VelocityPath=0.093; Kuka.CurrentCDSetIndex=0; Kuka.MovementParameterFieldEnabled=True; IlfCommand=LIN
;ENDFOLD
$BWDSTART = FALSE
LDAT_ACT=LCPDATP124
FDAT_ACT=FP124
BAS (#CP_PARAMS,0.093)
SET_CD_PARAMS (0)
LIN XP124 C_DIS

;ENDFOLD
;FOLD LIN P125 CONT Vel=0.093 m/s CPDATP125 Tool[2] Base[9] ;%{PE}
;FOLD Parameters ;%{h}
;Params IlfProvider=kukaroboter.basistech.inlineforms.movement.old; Kuka.IsGlobalPoint=False; Kuka.PointName=P125; Kuka.BlendingEnabled=TRUE; Kuka.MoveDataName=CPDATP125; Kuka.VelocityPath=0.093; Kuka.CurrentCDSetIndex=0; Kuka.MovementParameterFieldEnabled=True; IlfCommand=LIN
;ENDFOLD
$BWDSTART = FALSE
LDAT_ACT=LCPDATP125
FDAT_ACT=FP125
BAS (#CP_PARAMS,0.093)
SET_CD_PARAMS (0)
LIN XP125 C_DIS

;ENDFOLD
;FOLD LIN P126 CONT Vel=0.072 m/s CPDATP126 Tool[2] Base[9] ;%{PE}
;FOLD Parameters ;%{h}
;Params IlfProvider=kukaroboter.basistech.inlineforms.movement.old; Kuka.IsGlobalPoint=False; Kuka.PointName=P126; Kuka.BlendingEnabled=TRUE; Kuka.MoveDataName=CPDATP126; Kuka.VelocityPath=0.072; Kuka.CurrentCDSetIndex=0; Kuka.MovementParameterFieldEnabled=True; IlfCommand=LIN
;ENDFOLD
$BWDSTART = FALSE
LDAT_ACT=LCPDATP126
FDAT_ACT=FP126
BAS (#CP_PARAMS,0.072)
SET_CD_PARAMS (0)
LIN XP126 C_DIS

;ENDFOLD
;FOLD LIN P127 CONT Vel=0.072 m/s CPDATP127 Tool[2] Base[9] ;%{PE}
;FOLD Parameters ;%{h}
;Params IlfProvider=kukaroboter.basistech.inlineforms.movement.old; Kuka.IsGlobalPoint=False; Kuka.PointName=P127; Kuka.BlendingEnabled=TRUE; Kuka.MoveDataName=CPDATP127; Kuka.VelocityPath=0.072; Kuka.CurrentCDSetIndex=0; Kuka.MovementParameterFieldEnabled=True; IlfCommand=LIN
;ENDFOLD
$BWDSTART = FALSE
LDAT_ACT=LCPDATP127
FDAT_ACT=FP127
BAS (#CP_PARAMS,0.072)
SET_CD_PARAMS (0)
LIN XP127 C_DIS

;ENDFOLD
;FOLD LIN P128 CONT Vel=0.072 m/s CPDATP128 Tool[2] Base[9] ;%{PE}
;FOLD Parameters ;%{h}
;Params IlfProvider=kukaroboter.basistech.inlineforms.movement.old; Kuka.IsGlobalPoint=False; Kuka.PointName=P128; Kuka.BlendingEnabled=TRUE; Kuka.MoveDataName=CPDATP128; Kuka.VelocityPath=0.072; Kuka.CurrentCDSetIndex=0; Kuka.MovementParameterFieldEnabled=True; IlfCommand=LIN
;ENDFOLD
$BWDSTART = FALSE
LDAT_ACT=LCPDATP128
FDAT_ACT=FP128
BAS (#CP_PARAMS,0.072)
SET_CD_PARAMS (0)
LIN XP128 C_DIS

;ENDFOLD
;FOLD LIN P129 CONT Vel=0.072 m/s CPDATP129 Tool[2] Base[9] ;%{PE}
;FOLD Parameters ;%{h}
;Params IlfProvider=kukaroboter.basistech.inlineforms.movement.old; Kuka.IsGlobalPoint=False; Kuka.PointName=P129; Kuka.BlendingEnabled=TRUE; Kuka.MoveDataName=CPDATP129; Kuka.VelocityPath=0.072; Kuka.CurrentCDSetIndex=0; Kuka.MovementParameterFieldEnabled=True; IlfCommand=LIN
;ENDFOLD
$BWDSTART = FALSE
LDAT_ACT=LCPDATP129
FDAT_ACT=FP129
BAS (#CP_PARAMS,0.072)
SET_CD_PARAMS (0)
LIN XP129 C_DIS

;ENDFOLD
;FOLD LIN P130 CONT Vel=0.148 m/s CPDATP130 Tool[2] Base[9] ;%{PE}
;FOLD Parameters ;%{h}
;Params IlfProvider=kukaroboter.basistech.inlineforms.movement.old; Kuka.IsGlobalPoint=False; Kuka.PointName=P130; Kuka.BlendingEnabled=TRUE; Kuka.MoveDataName=CPDATP130; Kuka.VelocityPath=0.148; Kuka.CurrentCDSetIndex=0; Kuka.MovementParameterFieldEnabled=True; IlfCommand=LIN
;ENDFOLD
$BWDSTART = FALSE
LDAT_ACT=LCPDATP130
FDAT_ACT=FP130
BAS (#CP_PARAMS,0.148)
SET_CD_PARAMS (0)
LIN XP130 C_DIS

;ENDFOLD
;FOLD LIN P131 CONT Vel=0.148 m/s CPDATP131 Tool[2] Base[9] ;%{PE}
;FOLD Parameters ;%{h}
;Params IlfProvider=kukaroboter.basistech.inlineforms.movement.old; Kuka.IsGlobalPoint=False; Kuka.PointName=P131; Kuka.BlendingEnabled=TRUE; Kuka.MoveDataName=CPDATP131; Kuka.VelocityPath=0.148; Kuka.CurrentCDSetIndex=0; Kuka.MovementParameterFieldEnabled=True; IlfCommand=LIN
;ENDFOLD
$BWDSTART = FALSE
LDAT_ACT=LCPDATP131
FDAT_ACT=FP131
BAS (#CP_PARAMS,0.148)
SET_CD_PARAMS (0)
LIN XP131 C_DIS

;ENDFOLD
;FOLD LIN P132 CONT Vel=0.148 m/s CPDATP132 Tool[2] Base[9] ;%{PE}
;FOLD Parameters ;%{h}
;Params IlfProvider=kukaroboter.basistech.inlineforms.movement.old; Kuka.IsGlobalPoint=False; Kuka.PointName=P132; Kuka.BlendingEnabled=TRUE; Kuka.MoveDataName=CPDATP132; Kuka.VelocityPath=0.148; Kuka.CurrentCDSetIndex=0; Kuka.MovementParameterFieldEnabled=True; IlfCommand=LIN
;ENDFOLD
$BWDSTART = FALSE
LDAT_ACT=LCPDATP132
FDAT_ACT=FP132
BAS (#CP_PARAMS,0.148)
SET_CD_PARAMS (0)
LIN XP132 C_DIS

;ENDFOLD
;FOLD LIN P133 CONT Vel=0.148 m/s CPDATP133 Tool[2] Base[9] ;%{PE}
;FOLD Parameters ;%{h}
;Params IlfProvider=kukaroboter.basistech.inlineforms.movement.old; Kuka.IsGlobalPoint=False; Kuka.PointName=P133; Kuka.BlendingEnabled=TRUE; Kuka.MoveDataName=CPDATP133; Kuka.VelocityPath=0.148; Kuka.CurrentCDSetIndex=0; Kuka.MovementParameterFieldEnabled=True; IlfCommand=LIN
;ENDFOLD
$BWDSTART = FALSE
LDAT_ACT=LCPDATP133
FDAT_ACT=FP133
BAS (#CP_PARAMS,0.148)
SET_CD_PARAMS (0)
LIN XP133 C_DIS

;ENDFOLD
;FOLD LIN P134 CONT Vel=0.055 m/s CPDATP134 Tool[2] Base[9] ;%{PE}
;FOLD Parameters ;%{h}
;Params IlfProvider=kukaroboter.basistech.inlineforms.movement.old; Kuka.IsGlobalPoint=False; Kuka.PointName=P134; Kuka.BlendingEnabled=TRUE; Kuka.MoveDataName=CPDATP134; Kuka.VelocityPath=0.055; Kuka.CurrentCDSetIndex=0; Kuka.MovementParameterFieldEnabled=True; IlfCommand=LIN
;ENDFOLD
$BWDSTART = FALSE
LDAT_ACT=LCPDATP134
FDAT_ACT=FP134
BAS (#CP_PARAMS,0.055)
SET_CD_PARAMS (0)
LIN XP134 C_DIS

;ENDFOLD
;FOLD LIN P135 CONT Vel=0.055 m/s CPDATP135 Tool[2] Base[9] ;%{PE}
;FOLD Parameters ;%{h}
;Params IlfProvider=kukaroboter.basistech.inlineforms.movement.old; Kuka.IsGlobalPoint=False; Kuka.PointName=P135; Kuka.BlendingEnabled=TRUE; Kuka.MoveDataName=CPDATP135; Kuka.VelocityPath=0.055; Kuka.CurrentCDSetIndex=0; Kuka.MovementParameterFieldEnabled=True; IlfCommand=LIN
;ENDFOLD
$BWDSTART = FALSE
LDAT_ACT=LCPDATP135
FDAT_ACT=FP135
BAS (#CP_PARAMS,0.055)
SET_CD_PARAMS (0)
LIN XP135 C_DIS

;ENDFOLD
;FOLD LIN P136 CONT Vel=0.055 m/s CPDATP136 Tool[2] Base[9] ;%{PE}
;FOLD Parameters ;%{h}
;Params IlfProvider=kukaroboter.basistech.inlineforms.movement.old; Kuka.IsGlobalPoint=False; Kuka.PointName=P136; Kuka.BlendingEnabled=TRUE; Kuka.MoveDataName=CPDATP136; Kuka.VelocityPath=0.055; Kuka.CurrentCDSetIndex=0; Kuka.MovementParameterFieldEnabled=True; IlfCommand=LIN
;ENDFOLD
$BWDSTART = FALSE
LDAT_ACT=LCPDATP136
FDAT_ACT=FP136
BAS (#CP_PARAMS,0.055)
SET_CD_PARAMS (0)
LIN XP136 C_DIS

;ENDFOLD
;FOLD LIN P137 CONT Vel=0.055 m/s CPDATP137 Tool[2] Base[9] ;%{PE}
;FOLD Parameters ;%{h}
;Params IlfProvider=kukaroboter.basistech.inlineforms.movement.old; Kuka.IsGlobalPoint=False; Kuka.PointName=P137; Kuka.BlendingEnabled=TRUE; Kuka.MoveDataName=CPDATP137; Kuka.VelocityPath=0.055; Kuka.CurrentCDSetIndex=0; Kuka.MovementParameterFieldEnabled=True; IlfCommand=LIN
;ENDFOLD
$BWDSTART = FALSE
LDAT_ACT=LCPDATP137
FDAT_ACT=FP137
BAS (#CP_PARAMS,0.055)
SET_CD_PARAMS (0)
LIN XP137 C_DIS

;ENDFOLD
;FOLD LIN P138 CONT Vel=0.149 m/s CPDATP138 Tool[2] Base[9] ;%{PE}
;FOLD Parameters ;%{h}
;Params IlfProvider=kukaroboter.basistech.inlineforms.movement.old; Kuka.IsGlobalPoint=False; Kuka.PointName=P138; Kuka.BlendingEnabled=TRUE; Kuka.MoveDataName=CPDATP138; Kuka.VelocityPath=0.149; Kuka.CurrentCDSetIndex=0; Kuka.MovementParameterFieldEnabled=True; IlfCommand=LIN
;ENDFOLD
$BWDSTART = FALSE
LDAT_ACT=LCPDATP138
FDAT_ACT=FP138
BAS (#CP_PARAMS,0.149)
SET_CD_PARAMS (0)
LIN XP138 C_DIS

;ENDFOLD
;FOLD LIN P139 CONT Vel=0.149 m/s CPDATP139 Tool[2] Base[9] ;%{PE}
;FOLD Parameters ;%{h}
;Params IlfProvider=kukaroboter.basistech.inlineforms.movement.old; Kuka.IsGlobalPoint=False; Kuka.PointName=P139; Kuka.BlendingEnabled=TRUE; Kuka.MoveDataName=CPDATP139; Kuka.VelocityPath=0.149; Kuka.CurrentCDSetIndex=0; Kuka.MovementParameterFieldEnabled=True; IlfCommand=LIN
;ENDFOLD
$BWDSTART = FALSE
LDAT_ACT=LCPDATP139
FDAT_ACT=FP139
BAS (#CP_PARAMS,0.149)
SET_CD_PARAMS (0)
LIN XP139 C_DIS

;ENDFOLD
;FOLD LIN P140 CONT Vel=0.149 m/s CPDATP140 Tool[2] Base[9] ;%{PE}
;FOLD Parameters ;%{h}
;Params IlfProvider=kukaroboter.basistech.inlineforms.movement.old; Kuka.IsGlobalPoint=False; Kuka.PointName=P140; Kuka.BlendingEnabled=TRUE; Kuka.MoveDataName=CPDATP140; Kuka.VelocityPath=0.149; Kuka.CurrentCDSetIndex=0; Kuka.MovementParameterFieldEnabled=True; IlfCommand=LIN
;ENDFOLD
$BWDSTART = FALSE
LDAT_ACT=LCPDATP140
FDAT_ACT=FP140
BAS (#CP_PARAMS,0.149)
SET_CD_PARAMS (0)
LIN XP140 C_DIS

;ENDFOLD
;FOLD LIN P141 CONT Vel=0.149 m/s CPDATP141 Tool[2] Base[9] ;%{PE}
;FOLD Parameters ;%{h}
;Params IlfProvider=kukaroboter.basistech.inlineforms.movement.old; Kuka.IsGlobalPoint=False; Kuka.PointName=P141; Kuka.BlendingEnabled=TRUE; Kuka.MoveDataName=CPDATP141; Kuka.VelocityPath=0.149; Kuka.CurrentCDSetIndex=0; Kuka.MovementParameterFieldEnabled=True; IlfCommand=LIN
;ENDFOLD
$BWDSTART = FALSE
LDAT_ACT=LCPDATP141
FDAT_ACT=FP141
BAS (#CP_PARAMS,0.149)
SET_CD_PARAMS (0)
LIN XP141 C_DIS

;ENDFOLD
;FOLD LIN P142 CONT Vel=0.101 m/s CPDATP142 Tool[2] Base[9] ;%{PE}
;FOLD Parameters ;%{h}
;Params IlfProvider=kukaroboter.basistech.inlineforms.movement.old; Kuka.IsGlobalPoint=False; Kuka.PointName=P142; Kuka.BlendingEnabled=TRUE; Kuka.MoveDataName=CPDATP142; Kuka.VelocityPath=0.101; Kuka.CurrentCDSetIndex=0; Kuka.MovementParameterFieldEnabled=True; IlfCommand=LIN
;ENDFOLD
$BWDSTART = FALSE
LDAT_ACT=LCPDATP142
FDAT_ACT=FP142
BAS (#CP_PARAMS,0.101)
SET_CD_PARAMS (0)
LIN XP142 C_DIS

;ENDFOLD
;FOLD LIN P143 CONT Vel=0.101 m/s CPDATP143 Tool[2] Base[9] ;%{PE}
;FOLD Parameters ;%{h}
;Params IlfProvider=kukaroboter.basistech.inlineforms.movement.old; Kuka.IsGlobalPoint=False; Kuka.PointName=P143; Kuka.BlendingEnabled=TRUE; Kuka.MoveDataName=CPDATP143; Kuka.VelocityPath=0.101; Kuka.CurrentCDSetIndex=0; Kuka.MovementParameterFieldEnabled=True; IlfCommand=LIN
;ENDFOLD
$BWDSTART = FALSE
LDAT_ACT=LCPDATP143
FDAT_ACT=FP143
BAS (#CP_PARAMS,0.101)
SET_CD_PARAMS (0)
LIN XP143 C_DIS

;ENDFOLD
;FOLD LIN P144 CONT Vel=0.101 m/s CPDATP144 Tool[2] Base[9] ;%{PE}
;FOLD Parameters ;%{h}
;Params IlfProvider=kukaroboter.basistech.inlineforms.movement.old; Kuka.IsGlobalPoint=False; Kuka.PointName=P144; Kuka.BlendingEnabled=TRUE; Kuka.MoveDataName=CPDATP144; Kuka.VelocityPath=0.101; Kuka.CurrentCDSetIndex=0; Kuka.MovementParameterFieldEnabled=True; IlfCommand=LIN
;ENDFOLD
$BWDSTART = FALSE
LDAT_ACT=LCPDATP144
FDAT_ACT=FP144
BAS (#CP_PARAMS,0.101)
SET_CD_PARAMS (0)
LIN XP144 C_DIS

;ENDFOLD
;FOLD LIN P145 CONT Vel=0.101 m/s CPDATP145 Tool[2] Base[9] ;%{PE}
;FOLD Parameters ;%{h}
;Params IlfProvider=kukaroboter.basistech.inlineforms.movement.old; Kuka.IsGlobalPoint=False; Kuka.PointName=P145; Kuka.BlendingEnabled=TRUE; Kuka.MoveDataName=CPDATP145; Kuka.VelocityPath=0.101; Kuka.CurrentCDSetIndex=0; Kuka.MovementParameterFieldEnabled=True; IlfCommand=LIN
;ENDFOLD
$BWDSTART = FALSE
LDAT_ACT=LCPDATP145
FDAT_ACT=FP145
BAS (#CP_PARAMS,0.101)
SET_CD_PARAMS (0)
LIN XP145 C_DIS

;ENDFOLD
;FOLD LIN P146 CONT Vel=0.071 m/s CPDATP146 Tool[2] Base[9] ;%{PE}
;FOLD Parameters ;%{h}
;Params IlfProvider=kukaroboter.basistech.inlineforms.movement.old; Kuka.IsGlobalPoint=False; Kuka.PointName=P146; Kuka.BlendingEnabled=TRUE; Kuka.MoveDataName=CPDATP146; Kuka.VelocityPath=0.071; Kuka.CurrentCDSetIndex=0; Kuka.MovementParameterFieldEnabled=True; IlfCommand=LIN
;ENDFOLD
$BWDSTART = FALSE
LDAT_ACT=LCPDATP146
FDAT_ACT=FP146
BAS (#CP_PARAMS,0.071)
SET_CD_PARAMS (0)
LIN XP146 C_DIS

;ENDFOLD
;FOLD LIN P147 CONT Vel=0.071 m/s CPDATP147 Tool[2] Base[9] ;%{PE}
;FOLD Parameters ;%{h}
;Params IlfProvider=kukaroboter.basistech.inlineforms.movement.old; Kuka.IsGlobalPoint=False; Kuka.PointName=P147; Kuka.BlendingEnabled=TRUE; Kuka.MoveDataName=CPDATP147; Kuka.VelocityPath=0.071; Kuka.CurrentCDSetIndex=0; Kuka.MovementParameterFieldEnabled=True; IlfCommand=LIN
;ENDFOLD
$BWDSTART = FALSE
LDAT_ACT=LCPDATP147
FDAT_ACT=FP147
BAS (#CP_PARAMS,0.071)
SET_CD_PARAMS (0)
LIN XP147 C_DIS

;ENDFOLD
;FOLD LIN P148 CONT Vel=0.071 m/s CPDATP148 Tool[2] Base[9] ;%{PE}
;FOLD Parameters ;%{h}
;Params IlfProvider=kukaroboter.basistech.inlineforms.movement.old; Kuka.IsGlobalPoint=False; Kuka.PointName=P148; Kuka.BlendingEnabled=TRUE; Kuka.MoveDataName=CPDATP148; Kuka.VelocityPath=0.071; Kuka.CurrentCDSetIndex=0; Kuka.MovementParameterFieldEnabled=True; IlfCommand=LIN
;ENDFOLD
$BWDSTART = FALSE
LDAT_ACT=LCPDATP148
FDAT_ACT=FP148
BAS (#CP_PARAMS,0.071)
SET_CD_PARAMS (0)
LIN XP148 C_DIS

;ENDFOLD
;FOLD LIN P149 CONT Vel=0.071 m/s CPDATP149 Tool[2] Base[9] ;%{PE}
;FOLD Parameters ;%{h}
;Params IlfProvider=kukaroboter.basistech.inlineforms.movement.old; Kuka.IsGlobalPoint=False; Kuka.PointName=P149; Kuka.BlendingEnabled=TRUE; Kuka.MoveDataName=CPDATP149; Kuka.VelocityPath=0.071; Kuka.CurrentCDSetIndex=0; Kuka.MovementParameterFieldEnabled=True; IlfCommand=LIN
;ENDFOLD
$BWDSTART = FALSE
LDAT_ACT=LCPDATP149
FDAT_ACT=FP149
BAS (#CP_PARAMS,0.071)
SET_CD_PARAMS (0)
LIN XP149 C_DIS

;ENDFOLD
;FOLD LIN P150 CONT Vel=0.121 m/s CPDATP150 Tool[2] Base[9] ;%{PE}
;FOLD Parameters ;%{h}
;Params IlfProvider=kukaroboter.basistech.inlineforms.movement.old; Kuka.IsGlobalPoint=False; Kuka.PointName=P150; Kuka.BlendingEnabled=TRUE; Kuka.MoveDataName=CPDATP150; Kuka.VelocityPath=0.121; Kuka.CurrentCDSetIndex=0; Kuka.MovementParameterFieldEnabled=True; IlfCommand=LIN
;ENDFOLD
$BWDSTART = FALSE
LDAT_ACT=LCPDATP150
FDAT_ACT=FP150
BAS (#CP_PARAMS,0.121)
SET_CD_PARAMS (0)
LIN XP150 C_DIS

;ENDFOLD
;FOLD LIN P151 CONT Vel=0.121 m/s CPDATP151 Tool[2] Base[9] ;%{PE}
;FOLD Parameters ;%{h}
;Params IlfProvider=kukaroboter.basistech.inlineforms.movement.old; Kuka.IsGlobalPoint=False; Kuka.PointName=P151; Kuka.BlendingEnabled=TRUE; Kuka.MoveDataName=CPDATP151; Kuka.VelocityPath=0.121; Kuka.CurrentCDSetIndex=0; Kuka.MovementParameterFieldEnabled=True; IlfCommand=LIN
;ENDFOLD
$BWDSTART = FALSE
LDAT_ACT=LCPDATP151
FDAT_ACT=FP151
BAS (#CP_PARAMS,0.121)
SET_CD_PARAMS (0)
LIN XP151 C_DIS

;ENDFOLD
;FOLD LIN P152 CONT Vel=0.121 m/s CPDATP152 Tool[2] Base[9] ;%{PE}
;FOLD Parameters ;%{h}
;Params IlfProvider=kukaroboter.basistech.inlineforms.movement.old; Kuka.IsGlobalPoint=False; Kuka.PointName=P152; Kuka.BlendingEnabled=TRUE; Kuka.MoveDataName=CPDATP152; Kuka.VelocityPath=0.121; Kuka.CurrentCDSetIndex=0; Kuka.MovementParameterFieldEnabled=True; IlfCommand=LIN
;ENDFOLD
$BWDSTART = FALSE
LDAT_ACT=LCPDATP152
FDAT_ACT=FP152
BAS (#CP_PARAMS,0.121)
SET_CD_PARAMS (0)
LIN XP152 C_DIS

;ENDFOLD
;FOLD LIN P153 CONT Vel=0.121 m/s CPDATP153 Tool[2] Base[9] ;%{PE}
;FOLD Parameters ;%{h}
;Params IlfProvider=kukaroboter.basistech.inlineforms.movement.old; Kuka.IsGlobalPoint=False; Kuka.PointName=P153; Kuka.BlendingEnabled=TRUE; Kuka.MoveDataName=CPDATP153; Kuka.VelocityPath=0.121; Kuka.CurrentCDSetIndex=0; Kuka.MovementParameterFieldEnabled=True; IlfCommand=LIN
;ENDFOLD
$BWDSTART = FALSE
LDAT_ACT=LCPDATP153
FDAT_ACT=FP153
BAS (#CP_PARAMS,0.121)
SET_CD_PARAMS (0)
LIN XP153 C_DIS

;ENDFOLD
;FOLD LIN P154 CONT Vel=0.061 m/s CPDATP154 Tool[2] Base[9] ;%{PE}
;FOLD Parameters ;%{h}
;Params IlfProvider=kukaroboter.basistech.inlineforms.movement.old; Kuka.IsGlobalPoint=False; Kuka.PointName=P154; Kuka.BlendingEnabled=TRUE; Kuka.MoveDataName=CPDATP154; Kuka.VelocityPath=0.061; Kuka.CurrentCDSetIndex=0; Kuka.MovementParameterFieldEnabled=True; IlfCommand=LIN
;ENDFOLD
$BWDSTART = FALSE
LDAT_ACT=LCPDATP154
FDAT_ACT=FP154
BAS (#CP_PARAMS,0.061)
SET_CD_PARAMS (0)
LIN XP154 C_DIS

;ENDFOLD
;FOLD LIN P155 CONT Vel=0.061 m/s CPDATP155 Tool[2] Base[9] ;%{PE}
;FOLD Parameters ;%{h}
;Params IlfProvider=kukaroboter.basistech.inlineforms.movement.old; Kuka.IsGlobalPoint=False; Kuka.PointName=P155; Kuka.BlendingEnabled=TRUE; Kuka.MoveDataName=CPDATP155; Kuka.VelocityPath=0.061; Kuka.CurrentCDSetIndex=0; Kuka.MovementParameterFieldEnabled=True; IlfCommand=LIN
;ENDFOLD
$BWDSTART = FALSE
LDAT_ACT=LCPDATP155
FDAT_ACT=FP155
BAS (#CP_PARAMS,0.061)
SET_CD_PARAMS (0)
LIN XP155 C_DIS

;ENDFOLD
;FOLD LIN P156 CONT Vel=0.061 m/s CPDATP156 Tool[2] Base[9] ;%{PE}
;FOLD Parameters ;%{h}
;Params IlfProvider=kukaroboter.basistech.inlineforms.movement.old; Kuka.IsGlobalPoint=False; Kuka.PointName=P156; Kuka.BlendingEnabled=TRUE; Kuka.MoveDataName=CPDATP156; Kuka.VelocityPath=0.061; Kuka.CurrentCDSetIndex=0; Kuka.MovementParameterFieldEnabled=True; IlfCommand=LIN
;ENDFOLD
$BWDSTART = FALSE
LDAT_ACT=LCPDATP156
FDAT_ACT=FP156
BAS (#CP_PARAMS,0.061)
SET_CD_PARAMS (0)
LIN XP156 C_DIS

;ENDFOLD
;FOLD LIN P157 CONT Vel=0.061 m/s CPDATP157 Tool[2] Base[9] ;%{PE}
;FOLD Parameters ;%{h}
;Params IlfProvider=kukaroboter.basistech.inlineforms.movement.old; Kuka.IsGlobalPoint=False; Kuka.PointName=P157; Kuka.BlendingEnabled=TRUE; Kuka.MoveDataName=CPDATP157; Kuka.VelocityPath=0.061; Kuka.CurrentCDSetIndex=0; Kuka.MovementParameterFieldEnabled=True; IlfCommand=LIN
;ENDFOLD
$BWDSTART = FALSE
LDAT_ACT=LCPDATP157
FDAT_ACT=FP157
BAS (#CP_PARAMS,0.061)
SET_CD_PARAMS (0)
LIN XP157 C_DIS

;ENDFOLD
;FOLD LIN P158 CONT Vel=0.5 m/s CPDATP158 Tool[2] Base[9] ;%{PE}
;FOLD Parameters ;%{h}
;Params IlfProvider=kukaroboter.basistech.inlineforms.movement.old; Kuka.IsGlobalPoint=False; Kuka.PointName=P158; Kuka.BlendingEnabled=TRUE; Kuka.MoveDataName=CPDATP158; Kuka.VelocityPath=0.5; Kuka.CurrentCDSetIndex=0; Kuka.MovementParameterFieldEnabled=True; IlfCommand=LIN
;ENDFOLD
$BWDSTART = FALSE
LDAT_ACT=LCPDATP158
FDAT_ACT=FP158
BAS (#CP_PARAMS,0.5)
SET_CD_PARAMS (0)
LIN XP158 C_DIS

;ENDFOLD
;FOLD LIN P159 CONT Vel=1.0 m/s CPDATP159 Tool[2] Base[9] ;%{PE}
;FOLD Parameters ;%{h}
;Params IlfProvider=kukaroboter.basistech.inlineforms.movement.old; Kuka.IsGlobalPoint=False; Kuka.PointName=P159; Kuka.BlendingEnabled=TRUE; Kuka.MoveDataName=CPDATP159; Kuka.VelocityPath=1.0; Kuka.CurrentCDSetIndex=0; Kuka.MovementParameterFieldEnabled=True; IlfCommand=LIN
;ENDFOLD
$BWDSTART = FALSE
LDAT_ACT=LCPDATP159
FDAT_ACT=FP159
BAS (#CP_PARAMS,1.0)
SET_CD_PARAMS (0)
LIN XP159 C_DIS

;ENDFOLD
;FOLD LIN P160 CONT Vel=1.0 m/s CPDATP160 Tool[2] Base[9] ;%{PE}
;FOLD Parameters ;%{h}
;Params IlfProvider=kukaroboter.basistech.inlineforms.movement.old; Kuka.IsGlobalPoint=False; Kuka.PointName=P160; Kuka.BlendingEnabled=TRUE; Kuka.MoveDataName=CPDATP160; Kuka.VelocityPath=1.0; Kuka.CurrentCDSetIndex=0; Kuka.MovementParameterFieldEnabled=True; IlfCommand=LIN
;ENDFOLD
$BWDSTART = FALSE
LDAT_ACT=LCPDATP160
FDAT_ACT=FP160
BAS (#CP_PARAMS,1.0)
SET_CD_PARAMS (0)
LIN XP160 C_DIS

;ENDFOLD
END
;End of routine {i}

; --- Routine for substrate 2 ---
DEF Routine_2()
;FOLD LIN P161 CONT Vel=1.0 m/s CPDATP161 Tool[2] Base[8] ;%{PE}
;FOLD Parameters ;%{h}
;Params IlfProvider=kukaroboter.basistech.inlineforms.movement.old; Kuka.IsGlobalPoint=False; Kuka.PointName=P161; Kuka.BlendingEnabled=TRUE; Kuka.MoveDataName=CPDATP161; Kuka.VelocityPath=1.0; Kuka.CurrentCDSetIndex=0; Kuka.MovementParameterFieldEnabled=True; IlfCommand=LIN
;ENDFOLD
$BWDSTART = FALSE
LDAT_ACT=LCPDATP161
FDAT_ACT=FP161
BAS (#CP_PARAMS,1.0)
SET_CD_PARAMS (0)
LIN XP161 C_DIS

;ENDFOLD
;FOLD LIN P162 CONT Vel=0.123 m/s CPDATP162 Tool[2] Base[8] ;%{PE}
;FOLD Parameters ;%{h}
;Params IlfProvider=kukaroboter.basistech.inlineforms.movement.old; Kuka.IsGlobalPoint=False; Kuka.PointName=P162; Kuka.BlendingEnabled=TRUE; Kuka.MoveDataName=CPDATP162; Kuka.VelocityPath=0.123; Kuka.CurrentCDSetIndex=0; Kuka.MovementParameterFieldEnabled=True; IlfCommand=LIN
;ENDFOLD
$BWDSTART = FALSE
LDAT_ACT=LCPDATP162
FDAT_ACT=FP162
BAS (#CP_PARAMS,0.123)
SET_CD_PARAMS (0)
LIN XP162 C_DIS

;ENDFOLD
;FOLD LIN P163 CONT Vel=0.123 m/s CPDATP163 Tool[2] Base[8] ;%{PE}
;FOLD Parameters ;%{h}
;Params IlfProvider=kukaroboter.basistech.inlineforms.movement.old; Kuka.IsGlobalPoint=False; Kuka.PointName=P163; Kuka.BlendingEnabled=TRUE; Kuka.MoveDataName=CPDATP163; Kuka.VelocityPath=0.123; Kuka.CurrentCDSetIndex=0; Kuka.MovementParameterFieldEnabled=True; IlfCommand=LIN
;ENDFOLD
$BWDSTART = FALSE
LDAT_ACT=LCPDATP163
FDAT_ACT=FP163
BAS (#CP_PARAMS,0.123)
SET_CD_PARAMS (0)
LIN XP163 C_DIS

;ENDFOLD
;FOLD LIN P164 CONT Vel=0.123 m/s CPDATP164 Tool[2] Base[8] ;%{PE}
;FOLD Parameters ;%{h}
;Params IlfProvider=kukaroboter.basistech.inlineforms.movement.old; Kuka.IsGlobalPoint=False; Kuka.PointName=P164; Kuka.BlendingEnabled=TRUE; Kuka.MoveDataName=CPDATP164; Kuka.VelocityPath=0.123; Kuka.CurrentCDSetIndex=0; Kuka.MovementParameterFieldEnabled=True; IlfCommand=LIN
;ENDFOLD
$BWDSTART = FALSE
LDAT_ACT=LCPDATP164
FDAT_ACT=FP164
BAS (#CP_PARAMS,0.123)
SET_CD_PARAMS (0)
LIN XP164 C_DIS

;ENDFOLD
;FOLD LIN P165 CONT Vel=0.123 m/s CPDATP165 Tool[2] Base[8] ;%{PE}
;FOLD Parameters ;%{h}
;Params IlfProvider=kukaroboter.basistech.inlineforms.movement.old; Kuka.IsGlobalPoint=False; Kuka.PointName=P165; Kuka.BlendingEnabled=TRUE; Kuka.MoveDataName=CPDATP165; Kuka.VelocityPath=0.123; Kuka.CurrentCDSetIndex=0; Kuka.MovementParameterFieldEnabled=True; IlfCommand=LIN
;ENDFOLD
$BWDSTART = FALSE
LDAT_ACT=LCPDATP165
FDAT_ACT=FP165
BAS (#CP_PARAMS,0.123)
SET_CD_PARAMS (0)
LIN XP165 C_DIS

;ENDFOLD
;FOLD LIN P166 CONT Vel=0.128 m/s CPDATP166 Tool[2] Base[8] ;%{PE}
;FOLD Parameters ;%{h}
;Params IlfProvider=kukaroboter.basistech.inlineforms.movement.old; Kuka.IsGlobalPoint=False; Kuka.PointName=P166; Kuka.BlendingEnabled=TRUE; Kuka.MoveDataName=CPDATP166; Kuka.VelocityPath=0.128; Kuka.CurrentCDSetIndex=0; Kuka.MovementParameterFieldEnabled=True; IlfCommand=LIN
;ENDFOLD
$BWDSTART = FALSE
LDAT_ACT=LCPDATP166
FDAT_ACT=FP166
BAS (#CP_PARAMS,0.128)
SET_CD_PARAMS (0)
LIN XP166 C_DIS

;ENDFOLD
;FOLD LIN P167 CONT Vel=0.128 m/s CPDATP167 Tool[2] Base[8] ;%{PE}
;FOLD Parameters ;%{h}
;Params IlfProvider=kukaroboter.basistech.inlineforms.movement.old; Kuka.IsGlobalPoint=False; Kuka.PointName=P167; Kuka.BlendingEnabled=TRUE; Kuka.MoveDataName=CPDATP167; Kuka.VelocityPath=0.128; Kuka.CurrentCDSetIndex=0; Kuka.MovementParameterFieldEnabled=True; IlfCommand=LIN
;ENDFOLD
$BWDSTART = FALSE
LDAT_ACT=LCPDATP167
FDAT_ACT=FP167
BAS (#CP_PARAMS,0.128)
SET_CD_PARAMS (0)
LIN XP167 C_DIS

;ENDFOLD
;FOLD LIN P168 CONT Vel=0.128 m/s CPDATP168 Tool[2] Base[8] ;%{PE}
;FOLD Parameters ;%{h}
;Params IlfProvider=kukaroboter.basistech.inlineforms.movement.old; Kuka.IsGlobalPoint=False; Kuka.PointName=P168; Kuka.BlendingEnabled=TRUE; Kuka.MoveDataName=CPDATP168; Kuka.VelocityPath=0.128; Kuka.CurrentCDSetIndex=0; Kuka.MovementParameterFieldEnabled=True; IlfCommand=LIN
;ENDFOLD
$BWDSTART = FALSE
LDAT_ACT=LCPDATP168
FDAT_ACT=FP168
BAS (#CP_PARAMS,0.128)
SET_CD_PARAMS (0)
LIN XP168 C_DIS

;ENDFOLD
;FOLD LIN P169 CONT Vel=0.128 m/s CPDATP169 Tool[2] Base[8] ;%{PE}
;FOLD Parameters ;%{h}
;Params IlfProvider=kukaroboter.basistech.inlineforms.movement.old; Kuka.IsGlobalPoint=False; Kuka.PointName=P169; Kuka.BlendingEnabled=TRUE; Kuka.MoveDataName=CPDATP169; Kuka.VelocityPath=0.128; Kuka.CurrentCDSetIndex=0; Kuka.MovementParameterFieldEnabled=True; IlfCommand=LIN
;ENDFOLD
$BWDSTART = FALSE
LDAT_ACT=LCPDATP169
FDAT_ACT=FP169
BAS (#CP_PARAMS,0.128)
SET_CD_PARAMS (0)
LIN XP169 C_DIS

;ENDFOLD
;FOLD LIN P170 CONT Vel=0.103 m/s CPDATP170 Tool[2] Base[8] ;%{PE}
;FOLD Parameters ;%{h}
;Params IlfProvider=kukaroboter.basistech.inlineforms.movement.old; Kuka.IsGlobalPoint=False; Kuka.PointName=P170; Kuka.BlendingEnabled=TRUE; Kuka.MoveDataName=CPDATP170; Kuka.VelocityPath=0.103; Kuka.CurrentCDSetIndex=0; Kuka.MovementParameterFieldEnabled=True; IlfCommand=LIN
;ENDFOLD
$BWDSTART = FALSE
LDAT_ACT=LCPDATP170
FDAT_ACT=FP170
BAS (#CP_PARAMS,0.103)
SET_CD_PARAMS (0)
LIN XP170 C_DIS

;ENDFOLD
;FOLD LIN P171 CONT Vel=0.103 m/s CPDATP171 Tool[2] Base[8] ;%{PE}
;FOLD Parameters ;%{h}
;Params IlfProvider=kukaroboter.basistech.inlineforms.movement.old; Kuka.IsGlobalPoint=False; Kuka.PointName=P171; Kuka.BlendingEnabled=TRUE; Kuka.MoveDataName=CPDATP171; Kuka.VelocityPath=0.103; Kuka.CurrentCDSetIndex=0; Kuka.MovementParameterFieldEnabled=True; IlfCommand=LIN
;ENDFOLD
$BWDSTART = FALSE
LDAT_ACT=LCPDATP171
FDAT_ACT=FP171
BAS (#CP_PARAMS,0.103)
SET_CD_PARAMS (0)
LIN XP171 C_DIS

;ENDFOLD
;FOLD LIN P172 CONT Vel=0.103 m/s CPDATP172 Tool[2] Base[8] ;%{PE}
;FOLD Parameters ;%{h}
;Params IlfProvider=kukaroboter.basistech.inlineforms.movement.old; Kuka.IsGlobalPoint=False; Kuka.PointName=P172; Kuka.BlendingEnabled=TRUE; Kuka.MoveDataName=CPDATP172; Kuka.VelocityPath=0.103; Kuka.CurrentCDSetIndex=0; Kuka.MovementParameterFieldEnabled=True; IlfCommand=LIN
;ENDFOLD
$BWDSTART = FALSE
LDAT_ACT=LCPDATP172
FDAT_ACT=FP172
BAS (#CP_PARAMS,0.103)
SET_CD_PARAMS (0)
LIN XP172 C_DIS

;ENDFOLD
;FOLD LIN P173 CONT Vel=0.103 m/s CPDATP173 Tool[2] Base[8] ;%{PE}
;FOLD Parameters ;%{h}
;Params IlfProvider=kukaroboter.basistech.inlineforms.movement.old; Kuka.IsGlobalPoint=False; Kuka.PointName=P173; Kuka.BlendingEnabled=TRUE; Kuka.MoveDataName=CPDATP173; Kuka.VelocityPath=0.103; Kuka.CurrentCDSetIndex=0; Kuka.MovementParameterFieldEnabled=True; IlfCommand=LIN
;ENDFOLD
$BWDSTART = FALSE
LDAT_ACT=LCPDATP173
FDAT_ACT=FP173
BAS (#CP_PARAMS,0.103)
SET_CD_PARAMS (0)
LIN XP173 C_DIS

;ENDFOLD
;FOLD LIN P174 CONT Vel=0.108 m/s CPDATP174 Tool[2] Base[8] ;%{PE}
;FOLD Parameters ;%{h}
;Params IlfProvider=kukaroboter.basistech.inlineforms.movement.old; Kuka.IsGlobalPoint=False; Kuka.PointName=P174; Kuka.BlendingEnabled=TRUE; Kuka.MoveDataName=CPDATP174; Kuka.VelocityPath=0.108; Kuka.CurrentCDSetIndex=0; Kuka.MovementParameterFieldEnabled=True; IlfCommand=LIN
;ENDFOLD
$BWDSTART = FALSE
LDAT_ACT=LCPDATP174
FDAT_ACT=FP174
BAS (#CP_PARAMS,0.108)
SET_CD_PARAMS (0)
LIN XP174 C_DIS

;ENDFOLD
;FOLD LIN P175 CONT Vel=0.108 m/s CPDATP175 Tool[2] Base[8] ;%{PE}
;FOLD Parameters ;%{h}
;Params IlfProvider=kukaroboter.basistech.inlineforms.movement.old; Kuka.IsGlobalPoint=False; Kuka.PointName=P175; Kuka.BlendingEnabled=TRUE; Kuka.MoveDataName=CPDATP175; Kuka.VelocityPath=0.108; Kuka.CurrentCDSetIndex=0; Kuka.MovementParameterFieldEnabled=True; IlfCommand=LIN
;ENDFOLD
$BWDSTART = FALSE
LDAT_ACT=LCPDATP175
FDAT_ACT=FP175
BAS (#CP_PARAMS,0.108)
SET_CD_PARAMS (0)
LIN XP175 C_DIS

;ENDFOLD
;FOLD LIN P176 CONT Vel=0.108 m/s CPDATP176 Tool[2] Base[8] ;%{PE}
;FOLD Parameters ;%{h}
;Params IlfProvider=kukaroboter.basistech.inlineforms.movement.old; Kuka.IsGlobalPoint=False; Kuka.PointName=P176; Kuka.BlendingEnabled=TRUE; Kuka.MoveDataName=CPDATP176; Kuka.VelocityPath=0.108; Kuka.CurrentCDSetIndex=0; Kuka.MovementParameterFieldEnabled=True; IlfCommand=LIN
;ENDFOLD
$BWDSTART = FALSE
LDAT_ACT=LCPDATP176
FDAT_ACT=FP176
BAS (#CP_PARAMS,0.108)
SET_CD_PARAMS (0)
LIN XP176 C_DIS

;ENDFOLD
;FOLD LIN P177 CONT Vel=0.108 m/s CPDATP177 Tool[2] Base[8] ;%{PE}
;FOLD Parameters ;%{h}
;Params IlfProvider=kukaroboter.basistech.inlineforms.movement.old; Kuka.IsGlobalPoint=False; Kuka.PointName=P177; Kuka.BlendingEnabled=TRUE; Kuka.MoveDataName=CPDATP177; Kuka.VelocityPath=0.108; Kuka.CurrentCDSetIndex=0; Kuka.MovementParameterFieldEnabled=True; IlfCommand=LIN
;ENDFOLD
$BWDSTART = FALSE
LDAT_ACT=LCPDATP177
FDAT_ACT=FP177
BAS (#CP_PARAMS,0.108)
SET_CD_PARAMS (0)
LIN XP177 C_DIS

;ENDFOLD
;FOLD LIN P178 CONT Vel=0.095 m/s CPDATP178 Tool[2] Base[8] ;%{PE}
;FOLD Parameters ;%{h}
;Params IlfProvider=kukaroboter.basistech.inlineforms.movement.old; Kuka.IsGlobalPoint=False; Kuka.PointName=P178; Kuka.BlendingEnabled=TRUE; Kuka.MoveDataName=CPDATP178; Kuka.VelocityPath=0.095; Kuka.CurrentCDSetIndex=0; Kuka.MovementParameterFieldEnabled=True; IlfCommand=LIN
;ENDFOLD
$BWDSTART = FALSE
LDAT_ACT=LCPDATP178
FDAT_ACT=FP178
BAS (#CP_PARAMS,0.095)
SET_CD_PARAMS (0)
LIN XP178 C_DIS

;ENDFOLD
;FOLD LIN P179 CONT Vel=0.095 m/s CPDATP179 Tool[2] Base[8] ;%{PE}
;FOLD Parameters ;%{h}
;Params IlfProvider=kukaroboter.basistech.inlineforms.movement.old; Kuka.IsGlobalPoint=False; Kuka.PointName=P179; Kuka.BlendingEnabled=TRUE; Kuka.MoveDataName=CPDATP179; Kuka.VelocityPath=0.095; Kuka.CurrentCDSetIndex=0; Kuka.MovementParameterFieldEnabled=True; IlfCommand=LIN
;ENDFOLD
$BWDSTART = FALSE
LDAT_ACT=LCPDATP179
FDAT_ACT=FP179
BAS (#CP_PARAMS,0.095)
SET_CD_PARAMS (0)
LIN XP179 C_DIS

;ENDFOLD
;FOLD LIN P180 CONT Vel=0.095 m/s CPDATP180 Tool[2] Base[8] ;%{PE}
;FOLD Parameters ;%{h}
;Params IlfProvider=kukaroboter.basistech.inlineforms.movement.old; Kuka.IsGlobalPoint=False; Kuka.PointName=P180; Kuka.BlendingEnabled=TRUE; Kuka.MoveDataName=CPDATP180; Kuka.VelocityPath=0.095; Kuka.CurrentCDSetIndex=0; Kuka.MovementParameterFieldEnabled=True; IlfCommand=LIN
;ENDFOLD
$BWDSTART = FALSE
LDAT_ACT=LCPDATP180
FDAT_ACT=FP180
BAS (#CP_PARAMS,0.095)
SET_CD_PARAMS (0)
LIN XP180 C_DIS

;ENDFOLD
;FOLD LIN P181 CONT Vel=0.095 m/s CPDATP181 Tool[2] Base[8] ;%{PE}
;FOLD Parameters ;%{h}
;Params IlfProvider=kukaroboter.basistech.inlineforms.movement.old; Kuka.IsGlobalPoint=False; Kuka.PointName=P181; Kuka.BlendingEnabled=TRUE; Kuka.MoveDataName=CPDATP181; Kuka.VelocityPath=0.095; Kuka.CurrentCDSetIndex=0; Kuka.MovementParameterFieldEnabled=True; IlfCommand=LIN
;ENDFOLD
$BWDSTART = FALSE
LDAT_ACT=LCPDATP181
FDAT_ACT=FP181
BAS (#CP_PARAMS,0.095)
SET_CD_PARAMS (0)
LIN XP181 C_DIS

;ENDFOLD
;FOLD LIN P182 CONT Vel=0.142 m/s CPDATP182 Tool[2] Base[8] ;%{PE}
;FOLD Parameters ;%{h}
;Params IlfProvider=kukaroboter.basistech.inlineforms.movement.old; Kuka.IsGlobalPoint=False; Kuka.PointName=P182; Kuka.BlendingEnabled=TRUE; Kuka.MoveDataName=CPDATP182; Kuka.VelocityPath=0.142; Kuka.CurrentCDSetIndex=0; Kuka.MovementParameterFieldEnabled=True; IlfCommand=LIN
;ENDFOLD
$BWDSTART = FALSE
LDAT_ACT=LCPDATP182
FDAT_ACT=FP182
BAS (#CP_PARAMS,0.142)
SET_CD_PARAMS (0)
LIN XP182 C_DIS

;ENDFOLD
;FOLD LIN P183 CONT Vel=0.142 m/s CPDATP183 Tool[2] Base[8] ;%{PE}
;FOLD Parameters ;%{h}
;Params IlfProvider=kukaroboter.basistech.inlineforms.movement.old; Kuka.IsGlobalPoint=False; Kuka.PointName=P183; Kuka.BlendingEnabled=TRUE; Kuka.MoveDataName=CPDATP183; Kuka.VelocityPath=0.142; Kuka.CurrentCDSetIndex=0; Kuka.MovementParameterFieldEnabled=True; IlfCommand=LIN
;ENDFOLD
$BWDSTART = FALSE
LDAT_ACT=LCPDATP183
FDAT_ACT=FP183
BAS (#CP_PARAMS,0.142)
SET_CD_PARAMS (0)
LIN XP183 C_DIS

;ENDFOLD
;FOLD LIN P184 CONT Vel=0.142 m/s CPDATP184 Tool[2] Base[8] ;%{PE}
;FOLD Parameters ;%{h}
;Params IlfProvider=kukaroboter.basistech.inlineforms.movement.old; Kuka.IsGlobalPoint=False; Kuka.PointName=P184; Kuka.BlendingEnabled=TRUE; Kuka.MoveDataName=CPDATP184; Kuka.VelocityPath=0.142; Kuka.CurrentCDSetIndex=0; Kuka.MovementParameterFieldEnabled=True; IlfCommand=LIN
;ENDFOLD
$BWDSTART = FALSE
LDAT_ACT=LCPDATP184
FDAT_ACT=FP184
BAS (#CP_PARAMS,0.142)
SET_CD_PARAMS (0)
LIN XP184 C_DIS

;ENDFOLD
;FOLD LIN P185 CONT Vel=0.142 m/s CPDATP185 Tool[2] Base[8] ;%{PE}
;FOLD Parameters ;%{h}
;Params IlfProvider=kukaroboter.basistech.inlineforms.movement.old; Kuka.IsGlobalPoint=False; Kuka.PointName=P185; Kuka.BlendingEnabled=TRUE; Kuka.MoveDataName=CPDATP185; Kuka.VelocityPath=0.142; Kuka.CurrentCDSetIndex=0; Kuka.MovementParameterFieldEnabled=True; IlfCommand=LIN
;ENDFOLD
$BWDSTART = FALSE
LDAT_ACT=LCPDATP185
FDAT_ACT=FP185
BAS (#CP_PARAMS,0.142)
SET_CD_PARAMS (0)
LIN XP185 C_DIS

;ENDFOLD
;FOLD LIN P186 CONT Vel=0.142 m/s CPDATP186 Tool[2] Base[8] ;%{PE}
;FOLD Parameters ;%{h}
;Params IlfProvider=kukaroboter.basistech.inlineforms.movement.old; Kuka.IsGlobalPoint=False; Kuka.PointName=P186; Kuka.BlendingEnabled=TRUE; Kuka.MoveDataName=CPDATP186; Kuka.VelocityPath=0.142; Kuka.CurrentCDSetIndex=0; Kuka.MovementParameterFieldEnabled=True; IlfCommand=LIN
;ENDFOLD
$BWDSTART = FALSE
LDAT_ACT=LCPDATP186
FDAT_ACT=FP186
BAS (#CP_PARAMS,0.142)
SET_CD_PARAMS (0)
LIN XP186 C_DIS

;ENDFOLD
;FOLD LIN P187 CONT Vel=0.142 m/s CPDATP187 Tool[2] Base[8] ;%{PE}
;FOLD Parameters ;%{h}
;Params IlfProvider=kukaroboter.basistech.inlineforms.movement.old; Kuka.IsGlobalPoint=False; Kuka.PointName=P187; Kuka.BlendingEnabled=TRUE; Kuka.MoveDataName=CPDATP187; Kuka.VelocityPath=0.142; Kuka.CurrentCDSetIndex=0; Kuka.MovementParameterFieldEnabled=True; IlfCommand=LIN
;ENDFOLD
$BWDSTART = FALSE
LDAT_ACT=LCPDATP187
FDAT_ACT=FP187
BAS (#CP_PARAMS,0.142)
SET_CD_PARAMS (0)
LIN XP187 C_DIS

;ENDFOLD
;FOLD LIN P188 CONT Vel=0.142 m/s CPDATP188 Tool[2] Base[8] ;%{PE}
;FOLD Parameters ;%{h}
;Params IlfProvider=kukaroboter.basistech.inlineforms.movement.old; Kuka.IsGlobalPoint=False; Kuka.PointName=P188; Kuka.BlendingEnabled=TRUE; Kuka.MoveDataName=CPDATP188; Kuka.VelocityPath=0.142; Kuka.CurrentCDSetIndex=0; Kuka.MovementParameterFieldEnabled=True; IlfCommand=LIN
;ENDFOLD
$BWDSTART = FALSE
LDAT_ACT=LCPDATP188
FDAT_ACT=FP188
BAS (#CP_PARAMS,0.142)
SET_CD_PARAMS (0)
LIN XP188 C_DIS

;ENDFOLD
;FOLD LIN P189 CONT Vel=0.142 m/s CPDATP189 Tool[2] Base[8] ;%{PE}
;FOLD Parameters ;%{h}
;Params IlfProvider=kukaroboter.basistech.inlineforms.movement.old; Kuka.IsGlobalPoint=False; Kuka.PointName=P189; Kuka.BlendingEnabled=TRUE; Kuka.MoveDataName=CPDATP189; Kuka.VelocityPath=0.142; Kuka.CurrentCDSetIndex=0; Kuka.MovementParameterFieldEnabled=True; IlfCommand=LIN
;ENDFOLD
$BWDSTART = FALSE
LDAT_ACT=LCPDATP189
FDAT_ACT=FP189
BAS (#CP_PARAMS,0.142)
SET_CD_PARAMS (0)
LIN XP189 C_DIS

;ENDFOLD
;FOLD LIN P190 CONT Vel=0.064 m/s CPDATP190 Tool[2] Base[8] ;%{PE}
;FOLD Parameters ;%{h}
;Params IlfProvider=kukaroboter.basistech.inlineforms.movement.old; Kuka.IsGlobalPoint=False; Kuka.PointName=P190; Kuka.BlendingEnabled=TRUE; Kuka.MoveDataName=CPDATP190; Kuka.VelocityPath=0.064; Kuka.CurrentCDSetIndex=0; Kuka.MovementParameterFieldEnabled=True; IlfCommand=LIN
;ENDFOLD
$BWDSTART = FALSE
LDAT_ACT=LCPDATP190
FDAT_ACT=FP190
BAS (#CP_PARAMS,0.064)
SET_CD_PARAMS (0)
LIN XP190 C_DIS

;ENDFOLD
;FOLD LIN P191 CONT Vel=0.064 m/s CPDATP191 Tool[2] Base[8] ;%{PE}
;FOLD Parameters ;%{h}
;Params IlfProvider=kukaroboter.basistech.inlineforms.movement.old; Kuka.IsGlobalPoint=False; Kuka.PointName=P191; Kuka.BlendingEnabled=TRUE; Kuka.MoveDataName=CPDATP191; Kuka.VelocityPath=0.064; Kuka.CurrentCDSetIndex=0; Kuka.MovementParameterFieldEnabled=True; IlfCommand=LIN
;ENDFOLD
$BWDSTART = FALSE
LDAT_ACT=LCPDATP191
FDAT_ACT=FP191
BAS (#CP_PARAMS,0.064)
SET_CD_PARAMS (0)
LIN XP191 C_DIS

;ENDFOLD
;FOLD LIN P192 CONT Vel=0.064 m/s CPDATP192 Tool[2] Base[8] ;%{PE}
;FOLD Parameters ;%{h}
;Params IlfProvider=kukaroboter.basistech.inlineforms.movement.old; Kuka.IsGlobalPoint=False; Kuka.PointName=P192; Kuka.BlendingEnabled=TRUE; Kuka.MoveDataName=CPDATP192; Kuka.VelocityPath=0.064; Kuka.CurrentCDSetIndex=0; Kuka.MovementParameterFieldEnabled=True; IlfCommand=LIN
;ENDFOLD
$BWDSTART = FALSE
LDAT_ACT=LCPDATP192
FDAT_ACT=FP192
BAS (#CP_PARAMS,0.064)
SET_CD_PARAMS (0)
LIN XP192 C_DIS

;ENDFOLD
;FOLD LIN P193 CONT Vel=0.064 m/s CPDATP193 Tool[2] Base[8] ;%{PE}
;FOLD Parameters ;%{h}
;Params IlfProvider=kukaroboter.basistech.inlineforms.movement.old; Kuka.IsGlobalPoint=False; Kuka.PointName=P193; Kuka.BlendingEnabled=TRUE; Kuka.MoveDataName=CPDATP193; Kuka.VelocityPath=0.064; Kuka.CurrentCDSetIndex=0; Kuka.MovementParameterFieldEnabled=True; IlfCommand=LIN
;ENDFOLD
$BWDSTART = FALSE
LDAT_ACT=LCPDATP193
FDAT_ACT=FP193
BAS (#CP_PARAMS,0.064)
SET_CD_PARAMS (0)
LIN XP193 C_DIS

;ENDFOLD
;FOLD LIN P194 CONT Vel=0.055 m/s CPDATP194 Tool[2] Base[8] ;%{PE}
;FOLD Parameters ;%{h}
;Params IlfProvider=kukaroboter.basistech.inlineforms.movement.old; Kuka.IsGlobalPoint=False; Kuka.PointName=P194; Kuka.BlendingEnabled=TRUE; Kuka.MoveDataName=CPDATP194; Kuka.VelocityPath=0.055; Kuka.CurrentCDSetIndex=0; Kuka.MovementParameterFieldEnabled=True; IlfCommand=LIN
;ENDFOLD
$BWDSTART = FALSE
LDAT_ACT=LCPDATP194
FDAT_ACT=FP194
BAS (#CP_PARAMS,0.055)
SET_CD_PARAMS (0)
LIN XP194 C_DIS

;ENDFOLD
;FOLD LIN P195 CONT Vel=0.055 m/s CPDATP195 Tool[2] Base[8] ;%{PE}
;FOLD Parameters ;%{h}
;Params IlfProvider=kukaroboter.basistech.inlineforms.movement.old; Kuka.IsGlobalPoint=False; Kuka.PointName=P195; Kuka.BlendingEnabled=TRUE; Kuka.MoveDataName=CPDATP195; Kuka.VelocityPath=0.055; Kuka.CurrentCDSetIndex=0; Kuka.MovementParameterFieldEnabled=True; IlfCommand=LIN
;ENDFOLD
$BWDSTART = FALSE
LDAT_ACT=LCPDATP195
FDAT_ACT=FP195
BAS (#CP_PARAMS,0.055)
SET_CD_PARAMS (0)
LIN XP195 C_DIS

;ENDFOLD
;FOLD LIN P196 CONT Vel=0.055 m/s CPDATP196 Tool[2] Base[8] ;%{PE}
;FOLD Parameters ;%{h}
;Params IlfProvider=kukaroboter.basistech.inlineforms.movement.old; Kuka.IsGlobalPoint=False; Kuka.PointName=P196; Kuka.BlendingEnabled=TRUE; Kuka.MoveDataName=CPDATP196; Kuka.VelocityPath=0.055; Kuka.CurrentCDSetIndex=0; Kuka.MovementParameterFieldEnabled=True; IlfCommand=LIN
;ENDFOLD
$BWDSTART = FALSE
LDAT_ACT=LCPDATP196
FDAT_ACT=FP196
BAS (#CP_PARAMS,0.055)
SET_CD_PARAMS (0)
LIN XP196 C_DIS

